  [3771] = {x=-41.457, y=32.468, z=44, rx=180, rz=-142.083, shoulder=lefty, elbow=epositive, wrist=wpositive, fatherId=fReference[0]}
  [3772] = {x=-40.218, y=31.503, z=44, rx=-180, rz=-142.07, shoulder=lefty, elbow=epositive, wrist=wpositive, fatherId=fReference[0]}
  [3773] = {x=-38.979, y=30.538, z=44, rx=-180, rz=-142.056, shoulder=lefty, elbow=epositive, wrist=wpositive, fatherId=fReference[0]}
  [3774] = {x=-37.74, y=29.572, z=44, rx=180, rz=-142.044, shoulder=lefty, elbow=epositive, wrist=wpositive, fatherId=fReference[0]}
  [3775] = {x=-36.502, y=28.606, z=44, rx=180, rz=-142.031, shoulder=lefty, elbow=epositive, wrist=wpositive, fatherId=fReference[0]}
  [3776] = {x=-35.263, y=27.639, z=44, rx=180, rz=-142.019, shoulder=lefty, elbow=epositive, wrist=wpositive, fatherId=fReference[0]}
  [3777] = {x=-34.025, y=26.672, z=44, rx=-180, rz=-142.007, shoulder=lefty, elbow=epositive, wrist=wpositive, fatherId=fReference[0]}
  [3778] = {x=-32.787, y=25.705, z=44, rx=-180, rz=-141.996, shoulder=lefty, elbow=epositive, wrist=wpositive, fatherId=fReference[0]}
  [3779] = {x=-31.549, y=24.738, z=44, rx=-180, rz=-141.985, shoulder=lefty, elbow=epositive, wrist=wpositive, fatherId=fReference[0]}
  [3780] = {x=-30.311, y=23.77, z=44, rx=180, rz=-141.975, shoulder=lefty, elbow=epositive, wrist=wpositive, fatherId=fReference[0]}
  [3781] = {x=-29.073, y=22.802, z=44, rx=-180, rz=-141.965, shoulder=lefty, elbow=epositive, wrist=wpositive, fatherId=fReference[0]}
  [3782] = {x=-27.835, y=21.834, z=44, rx=180, rz=-141.956, shoulder=lefty, elbow=epositive, wrist=wpositive, fatherId=fReference[0]}
  [3783] = {x=-26.597, y=20.865, z=44, rx=180, rz=-141.947, shoulder=lefty, elbow=epositive, wrist=wpositive, fatherId=fReference[0]}
  [3784] = {x=-25.36, y=19.896, z=44, rx=-180, rz=-141.938, shoulder=lefty, elbow=epositive, wrist=wpositive, fatherId=fReference[0]}
  [3785] = {x=-24.122, y=18.927, z=44, rx=-180, rz=-141.93, shoulder=lefty, elbow=epositive, wrist=wpositive, fatherId=fReference[0]}
  [3786] = {x=-22.885, y=17.958, z=44, rx=180, rz=-141.922, shoulder=lefty, elbow=epositive, wrist=wpositive, fatherId=fReference[0]}
  [3787] = {x=-21.647, y=16.988, z=44, rx=180, rz=-141.915, shoulder=lefty, elbow=epositive, wrist=wpositive, fatherId=fReference[0]}
  [3788] = {x=-20.41, y=16.019, z=44, rx=-180, rz=-141.908, shoulder=lefty, elbow=epositive, wrist=wpositive, fatherId=fReference[0]}
  [3789] = {x=-19.172, y=15.049, z=44, rx=-180, rz=-141.901, shoulder=lefty, elbow=epositive, wrist=wpositive, fatherId=fReference[0]}
  [3790] = {x=-17.935, y=14.079, z=44, rx=-180, rz=-141.895, shoulder=lefty, elbow=epositive, wrist=wpositive, fatherId=fReference[0]}
  [3791] = {x=-16.698, y=13.109, z=44, rx=180, rz=-141.889, shoulder=lefty, elbow=epositive, wrist=wpositive, fatherId=fReference[0]}
  [3792] = {x=-15.461, y=12.138, z=44, rx=-180, rz=-141.884, shoulder=lefty, elbow=epositive, wrist=wpositive, fatherId=fReference[0]}
  [3793] = {x=-14.224, y=11.168, z=44, rx=-180, rz=-141.879, shoulder=lefty, elbow=epositive, wrist=wpositive, fatherId=fReference[0]}
  [3794] = {x=-12.987, y=10.197, z=44, rx=-180, rz=-141.875, shoulder=lefty, elbow=epositive, wrist=wpositive, fatherId=fReference[0]}
  [3795] = {x=-11.75, y=9.226, z=44, rx=-180, rz=-141.871, shoulder=lefty, elbow=epositive, wrist=wpositive, fatherId=fReference[0]}
  [3796] = {x=-10.513, y=8.255, z=44, rx=180, rz=-141.867, shoulder=lefty, elbow=epositive, wrist=wpositive, fatherId=fReference[0]}
  [3797] = {x=-9.276, y=7.284, z=44, rx=-180, rz=-141.864, shoulder=lefty, elbow=epositive, wrist=wpositive, fatherId=fReference[0]}
  [3798] = {x=-8.039, y=6.313, z=44, rx=-180, rz=-141.862, shoulder=lefty, elbow=epositive, wrist=wpositive, fatherId=fReference[0]}
  [3799] = {x=-6.802, y=5.342, z=44, rx=-180, rz=-141.859, shoulder=lefty, elbow=epositive, wrist=wpositive, fatherId=fReference[0]}
  [3800] = {x=-5.565, y=4.37, z=44, rx=180, rz=-141.857, shoulder=lefty, elbow=epositive, wrist=wpositive, fatherId=fReference[0]}
  [3801] = {x=-4.328, y=3.399, z=44, rx=180, rz=-141.856, shoulder=lefty, elbow=epositive, wrist=wpositive, fatherId=fReference[0]}
  [3802] = {x=-3.091, y=2.427, z=44, rx=-180, rz=-141.855, shoulder=lefty, elbow=epositive, wrist=wpositive, fatherId=fReference[0]}
  [3803] = {x=-1.854, y=1.456, z=44, rx=180, rz=-141.854, shoulder=lefty, elbow=epositive, wrist=wpositive, fatherId=fReference[0]}
  [3804] = {x=-0.617, y=0.484, z=44, rx=180, rz=-141.854, shoulder=lefty, elbow=epositive, wrist=wpositive, fatherId=fReference[0]}
  [3805] = {x=0.62, y=-0.487, z=44, rx=-180, rz=-141.854, shoulder=lefty, elbow=epositive, wrist=wpositive, fatherId=fReference[0]}
  [3806] = {x=1.857, y=-1.459, z=44, rx=180, rz=-141.855, shoulder=lefty, elbow=epositive, wrist=wpositive, fatherId=fReference[0]}
  [3807] = {x=3.094, y=-2.43, z=44, rx=-180, rz=-141.856, shoulder=lefty, elbow=epositive, wrist=wpositive, fatherId=fReference[0]}
  [3808] = {x=4.331, y=-3.402, z=44, rx=180, rz=-141.857, shoulder=lefty, elbow=epositive, wrist=wpositive, fatherId=fReference[0]}
  [3809] = {x=5.568, y=-4.373, z=44, rx=-180, rz=-141.859, shoulder=lefty, elbow=epositive, wrist=wpositive, fatherId=fReference[0]}
  [3810] = {x=6.805, y=-5.345, z=44, rx=-180, rz=-141.862, shoulder=lefty, elbow=epositive, wrist=wpositive, fatherId=fReference[0]}
  [3811] = {x=8.043, y=-6.316, z=44, rx=-180, rz=-141.864, shoulder=lefty, elbow=epositive, wrist=wpositive, fatherId=fReference[0]}
  [3812] = {x=9.28, y=-7.287, z=44, rx=-180, rz=-141.867, shoulder=lefty, elbow=epositive, wrist=wpositive, fatherId=fReference[0]}
  [3813] = {x=10.517, y=-8.259, z=44, rx=180, rz=-141.871, shoulder=lefty, elbow=epositive, wrist=wpositive, fatherId=fReference[0]}
  [3814] = {x=11.754, y=-9.23, z=44, rx=180, rz=-141.875, shoulder=lefty, elbow=epositive, wrist=wpositive, fatherId=fReference[0]}
  [3815] = {x=12.992, y=-10.201, z=44, rx=-180, rz=-141.879, shoulder=lefty, elbow=epositive, wrist=wpositive, fatherId=fReference[0]}
  [3816] = {x=14.229, y=-11.172, z=44, rx=-180, rz=-141.884, shoulder=lefty, elbow=epositive, wrist=wpositive, fatherId=fReference[0]}
  [3817] = {x=15.467, y=-12.143, z=44, rx=-180, rz=-141.89, shoulder=lefty, elbow=epositive, wrist=wpositive, fatherId=fReference[0]}
  [3818] = {x=16.704, y=-13.113, z=44, rx=180, rz=-141.895, shoulder=lefty, elbow=epositive, wrist=wpositive, fatherId=fReference[0]}
  [3819] = {x=17.942, y=-14.084, z=44, rx=180, rz=-141.901, shoulder=lefty, elbow=epositive, wrist=wpositive, fatherId=fReference[0]}
  [3820] = {x=19.179, y=-15.054, z=44, rx=-180, rz=-141.908, shoulder=lefty, elbow=epositive, wrist=wpositive, fatherId=fReference[0]}
  [3821] = {x=20.417, y=-16.025, z=44, rx=180, rz=-141.915, shoulder=lefty, elbow=epositive, wrist=wpositive, fatherId=fReference[0]}
  [3822] = {x=21.655, y=-16.995, z=44, rx=-180, rz=-141.922, shoulder=lefty, elbow=epositive, wrist=wpositive, fatherId=fReference[0]}
  [3823] = {x=22.893, y=-17.965, z=44, rx=-180, rz=-141.93, shoulder=lefty, elbow=epositive, wrist=wpositive, fatherId=fReference[0]}
  [3824] = {x=24.131, y=-18.934, z=44, rx=-180, rz=-141.938, shoulder=lefty, elbow=epositive, wrist=wpositive, fatherId=fReference[0]}
  [3825] = {x=25.369, y=-19.904, z=44, rx=-180, rz=-141.947, shoulder=lefty, elbow=epositive, wrist=wpositive, fatherId=fReference[0]}
  [3826] = {x=26.607, y=-20.873, z=44, rx=180, rz=-141.956, shoulder=lefty, elbow=epositive, wrist=wpositive, fatherId=fReference[0]}
  [3827] = {x=27.846, y=-21.842, z=44, rx=-180, rz=-141.965, shoulder=lefty, elbow=epositive, wrist=wpositive, fatherId=fReference[0]}
  [3828] = {x=29.084, y=-22.811, z=44, rx=-180, rz=-141.975, shoulder=lefty, elbow=epositive, wrist=wpositive, fatherId=fReference[0]}
  [3829] = {x=30.323, y=-23.779, z=44, rx=180, rz=-141.986, shoulder=lefty, elbow=epositive, wrist=wpositive, fatherId=fReference[0]}
  [3830] = {x=31.561, y=-24.748, z=44, rx=-180, rz=-141.996, shoulder=lefty, elbow=epositive, wrist=wpositive, fatherId=fReference[0]}
  [3831] = {x=32.8, y=-25.716, z=44, rx=180, rz=-142.008, shoulder=lefty, elbow=epositive, wrist=wpositive, fatherId=fReference[0]}
  [3832] = {x=34.039, y=-26.683, z=44, rx=-180, rz=-142.019, shoulder=lefty, elbow=epositive, wrist=wpositive, fatherId=fReference[0]}
  [3833] = {x=35.278, y=-27.651, z=44, rx=-180, rz=-142.031, shoulder=lefty, elbow=epositive, wrist=wpositive, fatherId=fReference[0]}
  [3834] = {x=36.517, y=-28.618, z=44, rx=180, rz=-142.044, shoulder=lefty, elbow=epositive, wrist=wpositive, fatherId=fReference[0]}
  [3835] = {x=37.757, y=-29.585, z=44, rx=-180, rz=-142.057, shoulder=lefty, elbow=epositive, wrist=wpositive, fatherId=fReference[0]}
  [3836] = {x=38.996, y=-30.551, z=44, rx=-180, rz=-142.07, shoulder=lefty, elbow=epositive, wrist=wpositive, fatherId=fReference[0]}
  [3837] = {x=40.236, y=-31.517, z=44, rx=180, rz=-142.084, shoulder=lefty, elbow=epositive, wrist=wpositive, fatherId=fReference[0]}
  [3838] = {x=41.476, y=-32.483, z=44, rx=-180, rz=-142.098, shoulder=lefty, elbow=epositive, wrist=wpositive, fatherId=fReference[0]}
  [3839] = {x=42.715, y=-33.448, z=44, rx=-180, rz=-142.113, shoulder=lefty, elbow=epositive, wrist=wpositive, fatherId=fReference[0]}
  [3840] = {x=43.956, y=-34.413, z=44, rx=-180, rz=-142.128, shoulder=lefty, elbow=epositive, wrist=wpositive, fatherId=fReference[0]}
  [3841] = {x=45.196, y=-35.377, z=44, rx=180, rz=-142.143, shoulder=lefty, elbow=epositive, wrist=wpositive, fatherId=fReference[0]}
  [3842] = {x=46.436, y=-36.342, z=44, rx=-180, rz=-142.159, shoulder=lefty, elbow=epositive, wrist=wpositive, fatherId=fReference[0]}
  [3843] = {x=47.677, y=-37.305, z=44, rx=-180, rz=-142.175, shoulder=lefty, elbow=epositive, wrist=wpositive, fatherId=fReference[0]}
  [3844] = {x=48.917, y=-38.269, z=44, rx=180, rz=-142.192, shoulder=lefty, elbow=epositive, wrist=wpositive, fatherId=fReference[0]}
  [3845] = {x=50.158, y=-39.231, z=44, rx=-180, rz=-142.209, shoulder=lefty, elbow=epositive, wrist=wpositive, fatherId=fReference[0]}
  [3846] = {x=51.399, y=-40.194, z=44, rx=-180, rz=-142.227, shoulder=lefty, elbow=epositive, wrist=wpositive, fatherId=fReference[0]}
  [3847] = {x=52.641, y=-41.156, z=44, rx=-180, rz=-142.245, shoulder=lefty, elbow=epositive, wrist=wpositive, fatherId=fReference[0]}
  [3848] = {x=53.882, y=-42.117, z=44, rx=-180, rz=-142.263, shoulder=lefty, elbow=epositive, wrist=wpositive, fatherId=fReference[0]}
  [3849] = {x=55.124, y=-43.078, z=44, rx=180, rz=-142.282, shoulder=lefty, elbow=epositive, wrist=wpositive, fatherId=fReference[0]}
  [3850] = {x=56.366, y=-44.038, z=44, rx=-180, rz=-142.302, shoulder=lefty, elbow=epositive, wrist=wpositive, fatherId=fReference[0]}
  [3851] = {x=57.608, y=-44.998, z=44, rx=-180, rz=-142.321, shoulder=lefty, elbow=epositive, wrist=wpositive, fatherId=fReference[0]}
  [3852] = {x=58.85, y=-45.958, z=44, rx=-180, rz=-142.342, shoulder=lefty, elbow=epositive, wrist=wpositive, fatherId=fReference[0]}
  [3853] = {x=60.092, y=-46.916, z=44, rx=-180, rz=-142.362, shoulder=lefty, elbow=epositive, wrist=wpositive, fatherId=fReference[0]}
  [3854] = {x=61.335, y=-47.875, z=44, rx=-180, rz=-142.383, shoulder=lefty, elbow=epositive, wrist=wpositive, fatherId=fReference[0]}
  [3855] = {x=62.578, y=-48.832, z=44, rx=180, rz=-142.405, shoulder=lefty, elbow=epositive, wrist=wpositive, fatherId=fReference[0]}
  [3856] = {x=63.821, y=-49.79, z=44, rx=-180, rz=-142.427, shoulder=lefty, elbow=epositive, wrist=wpositive, fatherId=fReference[0]}
  [3857] = {x=65.064, y=-50.746, z=44, rx=-180, rz=-142.449, shoulder=lefty, elbow=epositive, wrist=wpositive, fatherId=fReference[0]}
  [3858] = {x=66.308, y=-51.702, z=44, rx=-180, rz=-142.472, shoulder=lefty, elbow=epositive, wrist=wpositive, fatherId=fReference[0]}
  [3859] = {x=67.551, y=-52.657, z=44, rx=-180, rz=-142.496, shoulder=lefty, elbow=epositive, wrist=wpositive, fatherId=fReference[0]}
  [3860] = {x=68.795, y=-53.612, z=44, rx=-180, rz=-142.519, shoulder=lefty, elbow=epositive, wrist=wpositive, fatherId=fReference[0]}
  [3861] = {x=70.04, y=-54.566, z=44, rx=-180, rz=-142.543, shoulder=lefty, elbow=epositive, wrist=wpositive, fatherId=fReference[0]}
  [3862] = {x=71.284, y=-55.519, z=44, rx=180, rz=-142.568, shoulder=lefty, elbow=epositive, wrist=wpositive, fatherId=fReference[0]}
  [3863] = {x=72.529, y=-56.472, z=44, rx=-180, rz=-142.593, shoulder=lefty, elbow=epositive, wrist=wpositive, fatherId=fReference[0]}
  [3864] = {x=73.774, y=-57.424, z=44, rx=180, rz=-142.619, shoulder=lefty, elbow=epositive, wrist=wpositive, fatherId=fReference[0]}
  [3865] = {x=75.019, y=-58.376, z=44, rx=-180, rz=-142.645, shoulder=lefty, elbow=epositive, wrist=wpositive, fatherId=fReference[0]}
  [3866] = {x=76.264, y=-59.326, z=44, rx=-180, rz=-142.671, shoulder=lefty, elbow=epositive, wrist=wpositive, fatherId=fReference[0]}
  [3867] = {x=77.51, y=-60.276, z=44, rx=-180, rz=-142.698, shoulder=lefty, elbow=epositive, wrist=wpositive, fatherId=fReference[0]}
  [3868] = {x=78.756, y=-61.226, z=44, rx=-180, rz=-142.725, shoulder=lefty, elbow=epositive, wrist=wpositive, fatherId=fReference[0]}
  [3869] = {x=80.002, y=-62.174, z=44, rx=180, rz=-142.753, shoulder=lefty, elbow=epositive, wrist=wpositive, fatherId=fReference[0]}
  [3870] = {x=81.249, y=-63.122, z=44, rx=180, rz=-142.781, shoulder=lefty, elbow=epositive, wrist=wpositive, fatherId=fReference[0]}
  [3871] = {x=82.496, y=-64.069, z=44, rx=180, rz=-142.81, shoulder=lefty, elbow=epositive, wrist=wpositive, fatherId=fReference[0]}
  [3872] = {x=83.743, y=-65.015, z=44, rx=-180, rz=-142.839, shoulder=lefty, elbow=epositive, wrist=wpositive, fatherId=fReference[0]}
  [3873] = {x=84.99, y=-65.961, z=44, rx=-180, rz=-142.868, shoulder=lefty, elbow=epositive, wrist=wpositive, fatherId=fReference[0]}
  [3874] = {x=86.238, y=-66.905, z=44, rx=180, rz=-142.898, shoulder=lefty, elbow=epositive, wrist=wpositive, fatherId=fReference[0]}
  [3875] = {x=87.486, y=-67.849, z=44, rx=-180, rz=-142.929, shoulder=lefty, elbow=epositive, wrist=wpositive, fatherId=fReference[0]}
  [3876] = {x=88.734, y=-68.792, z=44, rx=-180, rz=-142.96, shoulder=lefty, elbow=epositive, wrist=wpositive, fatherId=fReference[0]}
  [3877] = {x=89.982, y=-69.734, z=44, rx=-180, rz=-142.991, shoulder=lefty, elbow=epositive, wrist=wpositive, fatherId=fReference[0]}
  [3878] = {x=91.231, y=-70.676, z=44, rx=-180, rz=-143.023, shoulder=lefty, elbow=epositive, wrist=wpositive, fatherId=fReference[0]}
  [3879] = {x=92.48, y=-71.616, z=44, rx=180, rz=-143.055, shoulder=lefty, elbow=epositive, wrist=wpositive, fatherId=fReference[0]}
  [3880] = {x=93.73, y=-72.556, z=44, rx=-180, rz=-143.088, shoulder=lefty, elbow=epositive, wrist=wpositive, fatherId=fReference[0]}
  [3881] = {x=94.979, y=-73.495, z=44, rx=-180, rz=-143.121, shoulder=lefty, elbow=epositive, wrist=wpositive, fatherId=fReference[0]}
  [3882] = {x=96.23, y=-74.432, z=44, rx=-180, rz=-143.155, shoulder=lefty, elbow=epositive, wrist=wpositive, fatherId=fReference[0]}
  [3883] = {x=97.48, y=-75.369, z=44, rx=-180, rz=-143.189, shoulder=lefty, elbow=epositive, wrist=wpositive, fatherId=fReference[0]}
  [3884] = {x=98.731, y=-76.305, z=44, rx=-180, rz=-143.224, shoulder=lefty, elbow=epositive, wrist=wpositive, fatherId=fReference[0]}
  [3885] = {x=99.982, y=-77.24, z=44, rx=-180, rz=-143.259, shoulder=lefty, elbow=epositive, wrist=wpositive, fatherId=fReference[0]}
  [3886] = {x=101.233, y=-78.175, z=44, rx=-180, rz=-143.294, shoulder=lefty, elbow=epositive, wrist=wpositive, fatherId=fReference[0]}
  [3887] = {x=102.485, y=-79.108, z=44, rx=180, rz=-143.33, shoulder=lefty, elbow=epositive, wrist=wpositive, fatherId=fReference[0]}
  [3888] = {x=103.737, y=-80.04, z=44, rx=180, rz=-143.367, shoulder=lefty, elbow=epositive, wrist=wpositive, fatherId=fReference[0]}
  [3889] = {x=104.989, y=-80.971, z=44, rx=-180, rz=-143.404, shoulder=lefty, elbow=epositive, wrist=wpositive, fatherId=fReference[0]}
  [3890] = {x=106.242, y=-81.901, z=44, rx=180, rz=-143.441, shoulder=lefty, elbow=epositive, wrist=wpositive, fatherId=fReference[0]}
  [3891] = {x=107.495, y=-82.831, z=44, rx=-180, rz=-143.479, shoulder=lefty, elbow=epositive, wrist=wpositive, fatherId=fReference[0]}
  [3892] = {x=108.748, y=-83.759, z=44, rx=-180, rz=-143.517, shoulder=lefty, elbow=epositive, wrist=wpositive, fatherId=fReference[0]}
  [3893] = {x=110.002, y=-84.686, z=44, rx=-180, rz=-143.556, shoulder=lefty, elbow=epositive, wrist=wpositive, fatherId=fReference[0]}
  [3894] = {x=111.256, y=-85.612, z=44, rx=-180, rz=-143.596, shoulder=lefty, elbow=epositive, wrist=wpositive, fatherId=fReference[0]}
  [3895] = {x=112.511, y=-86.537, z=44, rx=-180, rz=-143.635, shoulder=lefty, elbow=epositive, wrist=wpositive, fatherId=fReference[0]}
  [3896] = {x=113.766, y=-87.461, z=44, rx=-180, rz=-143.676, shoulder=lefty, elbow=epositive, wrist=wpositive, fatherId=fReference[0]}
  [3897] = {x=115.021, y=-88.384, z=44, rx=180, rz=-143.716, shoulder=lefty, elbow=epositive, wrist=wpositive, fatherId=fReference[0]}
  [3898] = {x=116.277, y=-89.306, z=44, rx=-180, rz=-143.758, shoulder=lefty, elbow=epositive, wrist=wpositive, fatherId=fReference[0]}
  [3899] = {x=117.533, y=-90.227, z=44, rx=-180, rz=-143.799, shoulder=lefty, elbow=epositive, wrist=wpositive, fatherId=fReference[0]}
  [3900] = {x=118.789, y=-91.146, z=44, rx=180, rz=-143.842, shoulder=lefty, elbow=epositive, wrist=wpositive, fatherId=fReference[0]}
  [3901] = {x=120.046, y=-92.065, z=44, rx=-180, rz=-143.884, shoulder=lefty, elbow=epositive, wrist=wpositive, fatherId=fReference[0]}
  [3902] = {x=121.304, y=-92.982, z=44, rx=-180, rz=-143.927, shoulder=lefty, elbow=epositive, wrist=wpositive, fatherId=fReference[0]}
  [3903] = {x=122.561, y=-93.898, z=44, rx=-180, rz=-143.971, shoulder=lefty, elbow=epositive, wrist=wpositive, fatherId=fReference[0]}
  [3904] = {x=123.819, y=-94.813, z=44, rx=-180, rz=-144.015, shoulder=lefty, elbow=epositive, wrist=wpositive, fatherId=fReference[0]}
  [3905] = {x=125.078, y=-95.727, z=44, rx=180, rz=-144.06, shoulder=lefty, elbow=epositive, wrist=wpositive, fatherId=fReference[0]}
  [3906] = {x=126.337, y=-96.64, z=44, rx=180, rz=-144.105, shoulder=lefty, elbow=epositive, wrist=wpositive, fatherId=fReference[0]}
  [3907] = {x=127.596, y=-97.551, z=44, rx=-180, rz=-144.151, shoulder=lefty, elbow=epositive, wrist=wpositive, fatherId=fReference[0]}
  [3908] = {x=128.856, y=-98.461, z=44, rx=180, rz=-144.197, shoulder=lefty, elbow=epositive, wrist=wpositive, fatherId=fReference[0]}
  [3909] = {x=130.116, y=-99.37, z=44, rx=-180, rz=-144.243, shoulder=lefty, elbow=epositive, wrist=wpositive, fatherId=fReference[0]}
  [3910] = {x=131.376, y=-100.278, z=44, rx=-180, rz=-144.291, shoulder=lefty, elbow=epositive, wrist=wpositive, fatherId=fReference[0]}
  [3911] = {x=132.637, y=-101.185, z=44, rx=-180, rz=-144.338, shoulder=lefty, elbow=epositive, wrist=wpositive, fatherId=fReference[0]}
  [3912] = {x=133.899, y=-102.09, z=44, rx=180, rz=-144.386, shoulder=lefty, elbow=epositive, wrist=wpositive, fatherId=fReference[0]}
  [3913] = {x=135.161, y=-102.994, z=44, rx=-180, rz=-144.435, shoulder=lefty, elbow=epositive, wrist=wpositive, fatherId=fReference[0]}
  [3914] = {x=136.423, y=-103.896, z=44, rx=-180, rz=-144.484, shoulder=lefty, elbow=epositive, wrist=wpositive, fatherId=fReference[0]}
  [3915] = {x=137.686, y=-104.798, z=44, rx=-180, rz=-144.534, shoulder=lefty, elbow=epositive, wrist=wpositive, fatherId=fReference[0]}
  [3916] = {x=138.949, y=-105.698, z=44, rx=-180, rz=-144.584, shoulder=lefty, elbow=epositive, wrist=wpositive, fatherId=fReference[0]}
  [3917] = {x=140.213, y=-106.596, z=44, rx=-180, rz=-144.634, shoulder=lefty, elbow=epositive, wrist=wpositive, fatherId=fReference[0]}
  [3918] = {x=141.477, y=-107.494, z=44, rx=180, rz=-144.686, shoulder=lefty, elbow=epositive, wrist=wpositive, fatherId=fReference[0]}
  [3919] = {x=142.742, y=-108.389, z=44, rx=-180, rz=-144.737, shoulder=lefty, elbow=epositive, wrist=wpositive, fatherId=fReference[0]}
  [3920] = {x=144.007, y=-109.284, z=44, rx=-180, rz=-144.789, shoulder=lefty, elbow=epositive, wrist=wpositive, fatherId=fReference[0]}
  [3921] = {x=145.273, y=-110.177, z=44, rx=180, rz=-144.842, shoulder=lefty, elbow=epositive, wrist=wpositive, fatherId=fReference[0]}
  [3922] = {x=146.539, y=-111.069, z=44, rx=-180, rz=-144.895, shoulder=lefty, elbow=epositive, wrist=wpositive, fatherId=fReference[0]}
  [3923] = {x=147.806, y=-111.959, z=44, rx=180, rz=-144.949, shoulder=lefty, elbow=epositive, wrist=wpositive, fatherId=fReference[0]}
  [3924] = {x=149.073, y=-112.848, z=44, rx=-180, rz=-145.003, shoulder=lefty, elbow=epositive, wrist=wpositive, fatherId=fReference[0]}
  [3925] = {x=150.34, y=-113.736, z=44, rx=-180, rz=-145.058, shoulder=lefty, elbow=epositive, wrist=wpositive, fatherId=fReference[0]}
  [3926] = {x=151.608, y=-114.622, z=44, rx=-180, rz=-145.113, shoulder=lefty, elbow=epositive, wrist=wpositive, fatherId=fReference[0]}
  [3927] = {x=152.877, y=-115.506, z=44, rx=-180, rz=-145.169, shoulder=lefty, elbow=epositive, wrist=wpositive, fatherId=fReference[0]}
  [3928] = {x=154.146, y=-116.389, z=44, rx=180, rz=-145.225, shoulder=lefty, elbow=epositive, wrist=wpositive, fatherId=fReference[0]}
  [3929] = {x=155.416, y=-117.271, z=44, rx=180, rz=-145.282, shoulder=lefty, elbow=epositive, wrist=wpositive, fatherId=fReference[0]}
  [3930] = {x=156.686, y=-118.151, z=44, rx=-180, rz=-145.34, shoulder=lefty, elbow=epositive, wrist=wpositive, fatherId=fReference[0]}
  [3931] = {x=157.957, y=-119.03, z=44, rx=-180, rz=-145.398, shoulder=lefty, elbow=epositive, wrist=wpositive, fatherId=fReference[0]}
  [3932] = {x=159.228, y=-119.907, z=44, rx=180, rz=-145.456, shoulder=lefty, elbow=epositive, wrist=wpositive, fatherId=fReference[0]}
  [3933] = {x=160.5, y=-120.782, z=44, rx=-180, rz=-145.515, shoulder=lefty, elbow=epositive, wrist=wpositive, fatherId=fReference[0]}
  [3934] = {x=161.772, y=-121.656, z=44, rx=180, rz=-145.575, shoulder=lefty, elbow=epositive, wrist=wpositive, fatherId=fReference[0]}
  [3935] = {x=163.045, y=-122.529, z=44, rx=180, rz=-145.635, shoulder=lefty, elbow=epositive, wrist=wpositive, fatherId=fReference[0]}
  [3936] = {x=164.319, y=-123.4, z=44, rx=180, rz=-145.695, shoulder=lefty, elbow=epositive, wrist=wpositive, fatherId=fReference[0]}
  [3937] = {x=165.593, y=-124.269, z=44, rx=-180, rz=-145.756, shoulder=lefty, elbow=epositive, wrist=wpositive, fatherId=fReference[0]}
  [3938] = {x=166.867, y=-125.136, z=44, rx=-180, rz=-145.818, shoulder=lefty, elbow=epositive, wrist=wpositive, fatherId=fReference[0]}
  [3939] = {x=168.142, y=-126.002, z=44, rx=-180, rz=-145.88, shoulder=lefty, elbow=epositive, wrist=wpositive, fatherId=fReference[0]}
  [3940] = {x=169.418, y=-126.867, z=44, rx=180, rz=-145.943, shoulder=lefty, elbow=epositive, wrist=wpositive, fatherId=fReference[0]}
  [3941] = {x=170.695, y=-127.73, z=44, rx=-180, rz=-146.006, shoulder=lefty, elbow=epositive, wrist=wpositive, fatherId=fReference[0]}
  [3942] = {x=171.971, y=-128.591, z=44, rx=-180, rz=-146.07, shoulder=lefty, elbow=epositive, wrist=wpositive, fatherId=fReference[0]}
  [3943] = {x=173.249, y=-129.45, z=44, rx=180, rz=-146.135, shoulder=lefty, elbow=epositive, wrist=wpositive, fatherId=fReference[0]}
  [3944] = {x=174.527, y=-130.308, z=44, rx=180, rz=-146.2, shoulder=lefty, elbow=epositive, wrist=wpositive, fatherId=fReference[0]}
  [3945] = {x=175.806, y=-131.164, z=44, rx=-180, rz=-146.265, shoulder=lefty, elbow=epositive, wrist=wpositive, fatherId=fReference[0]}
  [3946] = {x=177.085, y=-132.018, z=44, rx=-180, rz=-146.331, shoulder=lefty, elbow=epositive, wrist=wpositive, fatherId=fReference[0]}
  [3947] = {x=178.365, y=-132.871, z=44, rx=180, rz=-146.398, shoulder=lefty, elbow=epositive, wrist=wpositive, fatherId=fReference[0]}
  [3948] = {x=179.645, y=-133.721, z=44, rx=-180, rz=-146.465, shoulder=lefty, elbow=epositive, wrist=wpositive, fatherId=fReference[0]}
  [3949] = {x=180.927, y=-134.571, z=44, rx=-180, rz=-146.533, shoulder=lefty, elbow=epositive, wrist=wpositive, fatherId=fReference[0]}
  [3950] = {x=182.208, y=-135.418, z=44, rx=-180, rz=-146.601, shoulder=lefty, elbow=epositive, wrist=wpositive, fatherId=fReference[0]}
  [3951] = {x=183.491, y=-136.263, z=44, rx=180, rz=-146.67, shoulder=lefty, elbow=epositive, wrist=wpositive, fatherId=fReference[0]}
  [3952] = {x=184.774, y=-137.107, z=44, rx=-180, rz=-146.74, shoulder=lefty, elbow=epositive, wrist=wpositive, fatherId=fReference[0]}
  [3953] = {x=186.057, y=-137.949, z=44, rx=-180, rz=-146.81, shoulder=lefty, elbow=epositive, wrist=wpositive, fatherId=fReference[0]}
  [3954] = {x=187.341, y=-138.789, z=44, rx=180, rz=-146.881, shoulder=lefty, elbow=epositive, wrist=wpositive, fatherId=fReference[0]}
  [3955] = {x=188.626, y=-139.627, z=44, rx=-180, rz=-146.952, shoulder=lefty, elbow=epositive, wrist=wpositive, fatherId=fReference[0]}
  [3956] = {x=189.912, y=-140.464, z=44, rx=-180, rz=-147.024, shoulder=lefty, elbow=epositive, wrist=wpositive, fatherId=fReference[0]}
  [3957] = {x=191.198, y=-141.298, z=44, rx=-180, rz=-147.096, shoulder=lefty, elbow=epositive, wrist=wpositive, fatherId=fReference[0]}
  [3958] = {x=192.485, y=-142.131, z=44, rx=-180, rz=-147.169, shoulder=lefty, elbow=epositive, wrist=wpositive, fatherId=fReference[0]}
  [3959] = {x=193.772, y=-142.961, z=44, rx=-180, rz=-147.243, shoulder=lefty, elbow=epositive, wrist=wpositive, fatherId=fReference[0]}
  [3960] = {x=195.06, y=-143.79, z=44, rx=-180, rz=-147.317, shoulder=lefty, elbow=epositive, wrist=wpositive, fatherId=fReference[0]}
  [3961] = {x=196.349, y=-144.617, z=44, rx=-180, rz=-147.392, shoulder=lefty, elbow=epositive, wrist=wpositive, fatherId=fReference[0]}
  [3962] = {x=197.639, y=-145.442, z=44, rx=-180, rz=-147.467, shoulder=lefty, elbow=epositive, wrist=wpositive, fatherId=fReference[0]}
  [3963] = {x=198.929, y=-146.265, z=44, rx=-180, rz=-147.543, shoulder=lefty, elbow=epositive, wrist=wpositive, fatherId=fReference[0]}
  [3964] = {x=200.219, y=-147.086, z=44, rx=-180, rz=-147.619, shoulder=lefty, elbow=epositive, wrist=wpositive, fatherId=fReference[0]}
  [3965] = {x=201.511, y=-147.905, z=44, rx=-180, rz=-147.697, shoulder=lefty, elbow=epositive, wrist=wpositive, fatherId=fReference[0]}
  [3966] = {x=202.803, y=-148.722, z=44, rx=-180, rz=-147.774, shoulder=lefty, elbow=epositive, wrist=wpositive, fatherId=fReference[0]}
  [3967] = {x=204.096, y=-149.536, z=44, rx=-180, rz=-147.853, shoulder=lefty, elbow=epositive, wrist=wpositive, fatherId=fReference[0]}
  [3968] = {x=205.389, y=-150.349, z=44, rx=-180, rz=-147.931, shoulder=lefty, elbow=epositive, wrist=wpositive, fatherId=fReference[0]}
  [3969] = {x=206.683, y=-151.16, z=44, rx=180, rz=-148.011, shoulder=lefty, elbow=epositive, wrist=wpositive, fatherId=fReference[0]}
  [3970] = {x=207.978, y=-151.969, z=44, rx=180, rz=-148.091, shoulder=lefty, elbow=epositive, wrist=wpositive, fatherId=fReference[0]}
  [3971] = {x=209.273, y=-152.775, z=44, rx=180, rz=-148.172, shoulder=lefty, elbow=epositive, wrist=wpositive, fatherId=fReference[0]}
  [3972] = {x=210.569, y=-153.58, z=44, rx=180, rz=-148.253, shoulder=lefty, elbow=epositive, wrist=wpositive, fatherId=fReference[0]}
  [3973] = {x=211.866, y=-154.382, z=44, rx=180, rz=-148.335, shoulder=lefty, elbow=epositive, wrist=wpositive, fatherId=fReference[0]}
  [3974] = {x=213.164, y=-155.183, z=44, rx=-180, rz=-148.418, shoulder=lefty, elbow=epositive, wrist=wpositive, fatherId=fReference[0]}
  [3975] = {x=214.462, y=-155.981, z=44, rx=-180, rz=-148.501, shoulder=lefty, elbow=epositive, wrist=wpositive, fatherId=fReference[0]}
  [3976] = {x=215.761, y=-156.777, z=44, rx=180, rz=-148.585, shoulder=lefty, elbow=epositive, wrist=wpositive, fatherId=fReference[0]}
  [3977] = {x=217.06, y=-157.57, z=44, rx=-180, rz=-148.669, shoulder=lefty, elbow=epositive, wrist=wpositive, fatherId=fReference[0]}
  [3978] = {x=218.361, y=-158.362, z=44, rx=-180, rz=-148.754, shoulder=lefty, elbow=epositive, wrist=wpositive, fatherId=fReference[0]}
  [3979] = {x=219.662, y=-159.151, z=44, rx=180, rz=-148.84, shoulder=lefty, elbow=epositive, wrist=wpositive, fatherId=fReference[0]}
  [3980] = {x=220.963, y=-159.938, z=44, rx=-180, rz=-148.926, shoulder=lefty, elbow=epositive, wrist=wpositive, fatherId=fReference[0]}
  [3981] = {x=222.266, y=-160.723, z=44, rx=-180, rz=-149.013, shoulder=lefty, elbow=epositive, wrist=wpositive, fatherId=fReference[0]}
  [3982] = {x=223.569, y=-161.506, z=44, rx=180, rz=-149.101, shoulder=lefty, elbow=epositive, wrist=wpositive, fatherId=fReference[0]}
  [3983] = {x=224.872, y=-162.286, z=44, rx=180, rz=-149.189, shoulder=lefty, elbow=epositive, wrist=wpositive, fatherId=fReference[0]}
  [3984] = {x=226.177, y=-163.064, z=44, rx=-180, rz=-149.278, shoulder=lefty, elbow=epositive, wrist=wpositive, fatherId=fReference[0]}
  [3985] = {x=227.482, y=-163.84, z=44, rx=-180, rz=-149.367, shoulder=lefty, elbow=epositive, wrist=wpositive, fatherId=fReference[0]}
  [3986] = {x=228.788, y=-164.613, z=44, rx=-180, rz=-149.458, shoulder=lefty, elbow=epositive, wrist=wpositive, fatherId=fReference[0]}
  [3987] = {x=230.095, y=-165.384, z=44, rx=-180, rz=-149.548, shoulder=lefty, elbow=epositive, wrist=wpositive, fatherId=fReference[0]}
  [3988] = {x=231.402, y=-166.152, z=44, rx=-180, rz=-149.64, shoulder=lefty, elbow=epositive, wrist=wpositive, fatherId=fReference[0]}
  [3989] = {x=232.71, y=-166.919, z=44, rx=-180, rz=-149.732, shoulder=lefty, elbow=epositive, wrist=wpositive, fatherId=fReference[0]}
  [3990] = {x=234.019, y=-167.682, z=44, rx=-180, rz=-149.824, shoulder=lefty, elbow=epositive, wrist=wpositive, fatherId=fReference[0]}
  [3991] = {x=235.328, y=-168.444, z=44, rx=-180, rz=-149.918, shoulder=lefty, elbow=epositive, wrist=wpositive, fatherId=fReference[0]}
  [3992] = {x=236.638, y=-169.203, z=44, rx=-180, rz=-150.012, shoulder=lefty, elbow=epositive, wrist=wpositive, fatherId=fReference[0]}
  [3993] = {x=237.949, y=-169.959, z=44, rx=-180, rz=-150.106, shoulder=lefty, elbow=epositive, wrist=wpositive, fatherId=fReference[0]}
  [3994] = {x=239.261, y=-170.713, z=44, rx=-180, rz=-150.202, shoulder=lefty, elbow=epositive, wrist=wpositive, fatherId=fReference[0]}
  [3995] = {x=240.573, y=-171.465, z=44, rx=-180, rz=-150.298, shoulder=lefty, elbow=epositive, wrist=wpositive, fatherId=fReference[0]}
  [3996] = {x=241.886, y=-172.214, z=44, rx=-180, rz=-150.394, shoulder=lefty, elbow=epositive, wrist=wpositive, fatherId=fReference[0]}
  [3997] = {x=243.2, y=-172.96, z=44, rx=-180, rz=-150.491, shoulder=lefty, elbow=epositive, wrist=wpositive, fatherId=fReference[0]}
  [3998] = {x=244.514, y=-173.704, z=44, rx=-180, rz=-150.589, shoulder=lefty, elbow=epositive, wrist=wpositive, fatherId=fReference[0]}
  [3999] = {x=245.83, y=-174.446, z=44, rx=-180, rz=-150.688, shoulder=lefty, elbow=epositive, wrist=wpositive, fatherId=fReference[0]}
  [4000] = {x=247.146, y=-175.184, z=44, rx=-180, rz=-150.787, shoulder=lefty, elbow=epositive, wrist=wpositive, fatherId=fReference[0]}
  [4001] = {x=248.462, y=-175.921, z=44, rx=180, rz=-150.887, shoulder=lefty, elbow=epositive, wrist=wpositive, fatherId=fReference[0]}
  [4002] = {x=249.78, y=-176.654, z=44, rx=-180, rz=-150.988, shoulder=lefty, elbow=epositive, wrist=wpositive, fatherId=fReference[0]}
  [4003] = {x=251.098, y=-177.385, z=44, rx=180, rz=-151.089, shoulder=lefty, elbow=epositive, wrist=wpositive, fatherId=fReference[0]}
  [4004] = {x=252.417, y=-178.114, z=44, rx=-180, rz=-151.191, shoulder=lefty, elbow=epositive, wrist=wpositive, fatherId=fReference[0]}
  [4005] = {x=253.736, y=-178.839, z=44, rx=-180, rz=-151.293, shoulder=lefty, elbow=epositive, wrist=wpositive, fatherId=fReference[0]}
  [4006] = {x=255.056, y=-179.562, z=44, rx=180, rz=-151.397, shoulder=lefty, elbow=epositive, wrist=wpositive, fatherId=fReference[0]}
  [4007] = {x=256.378, y=-180.283, z=44, rx=180, rz=-151.501, shoulder=lefty, elbow=epositive, wrist=wpositive, fatherId=fReference[0]}
  [4008] = {x=257.699, y=-181, z=44, rx=-180, rz=-151.605, shoulder=lefty, elbow=epositive, wrist=wpositive, fatherId=fReference[0]}
  [4009] = {x=259.022, y=-181.715, z=44, rx=180, rz=-151.711, shoulder=lefty, elbow=epositive, wrist=wpositive, fatherId=fReference[0]}
  [4010] = {x=260.345, y=-182.427, z=44, rx=-180, rz=-151.817, shoulder=lefty, elbow=epositive, wrist=wpositive, fatherId=fReference[0]}
  [4011] = {x=261.669, y=-183.137, z=44, rx=-180, rz=-151.923, shoulder=lefty, elbow=epositive, wrist=wpositive, fatherId=fReference[0]}
  [4012] = {x=262.994, y=-183.843, z=44, rx=180, rz=-152.031, shoulder=lefty, elbow=epositive, wrist=wpositive, fatherId=fReference[0]}
  [4013] = {x=264.319, y=-184.547, z=44, rx=-180, rz=-152.139, shoulder=lefty, elbow=epositive, wrist=wpositive, fatherId=fReference[0]}
  [4014] = {x=265.645, y=-185.248, z=44, rx=-180, rz=-152.247, shoulder=lefty, elbow=epositive, wrist=wpositive, fatherId=fReference[0]}
  [4015] = {x=266.972, y=-185.946, z=44, rx=180, rz=-152.357, shoulder=lefty, elbow=epositive, wrist=wpositive, fatherId=fReference[0]}
  [4016] = {x=268.3, y=-186.642, z=44, rx=180, rz=-152.467, shoulder=lefty, elbow=epositive, wrist=wpositive, fatherId=fReference[0]}
  [4017] = {x=269.628, y=-187.334, z=44, rx=180, rz=-152.578, shoulder=lefty, elbow=epositive, wrist=wpositive, fatherId=fReference[0]}
  [4018] = {x=270.957, y=-188.024, z=44, rx=-180, rz=-152.689, shoulder=lefty, elbow=epositive, wrist=wpositive, fatherId=fReference[0]}
  [4019] = {x=272.287, y=-188.711, z=44, rx=-180, rz=-152.801, shoulder=lefty, elbow=epositive, wrist=wpositive, fatherId=fReference[0]}
  [4020] = {x=273.617, y=-189.394, z=44, rx=180, rz=-152.914, shoulder=lefty, elbow=epositive, wrist=wpositive, fatherId=fReference[0]}
  [4021] = {x=274.948, y=-190.075, z=44, rx=-180, rz=-153.028, shoulder=lefty, elbow=epositive, wrist=wpositive, fatherId=fReference[0]}
  [4022] = {x=276.28, y=-190.753, z=44, rx=-180, rz=-153.142, shoulder=lefty, elbow=epositive, wrist=wpositive, fatherId=fReference[0]}
  [4023] = {x=277.613, y=-191.428, z=44, rx=-180, rz=-153.257, shoulder=lefty, elbow=epositive, wrist=wpositive, fatherId=fReference[0]}
  [4024] = {x=278.947, y=-192.1, z=44, rx=-180, rz=-153.372, shoulder=lefty, elbow=epositive, wrist=wpositive, fatherId=fReference[0]}
  [4025] = {x=280.281, y=-192.769, z=44, rx=-180, rz=-153.489, shoulder=lefty, elbow=epositive, wrist=wpositive, fatherId=fReference[0]}
  [4026] = {x=281.616, y=-193.435, z=44, rx=-180, rz=-153.606, shoulder=lefty, elbow=epositive, wrist=wpositive, fatherId=fReference[0]}
  [4027] = {x=282.951, y=-194.097, z=44, rx=-180, rz=-153.724, shoulder=lefty, elbow=epositive, wrist=wpositive, fatherId=fReference[0]}
  [4028] = {x=284.288, y=-194.757, z=44, rx=180, rz=-153.842, shoulder=lefty, elbow=epositive, wrist=wpositive, fatherId=fReference[0]}
  [4029] = {x=285.625, y=-195.414, z=44, rx=-180, rz=-153.961, shoulder=lefty, elbow=epositive, wrist=wpositive, fatherId=fReference[0]}
  [4030] = {x=286.963, y=-196.068, z=44, rx=180, rz=-154.081, shoulder=lefty, elbow=epositive, wrist=wpositive, fatherId=fReference[0]}
  [4031] = {x=288.301, y=-196.718, z=44, rx=-180, rz=-154.202, shoulder=lefty, elbow=epositive, wrist=wpositive, fatherId=fReference[0]}
  [4032] = {x=289.64, y=-197.365, z=44, rx=-180, rz=-154.323, shoulder=lefty, elbow=epositive, wrist=wpositive, fatherId=fReference[0]}
  [4033] = {x=290.98, y=-198.01, z=44, rx=180, rz=-154.445, shoulder=lefty, elbow=epositive, wrist=wpositive, fatherId=fReference[0]}
  [4034] = {x=292.321, y=-198.651, z=44, rx=-180, rz=-154.568, shoulder=lefty, elbow=epositive, wrist=wpositive, fatherId=fReference[0]}
  [4035] = {x=293.663, y=-199.289, z=44, rx=-180, rz=-154.691, shoulder=lefty, elbow=epositive, wrist=wpositive, fatherId=fReference[0]}
  [4036] = {x=295.005, y=-199.923, z=44, rx=-180, rz=-154.815, shoulder=lefty, elbow=epositive, wrist=wpositive, fatherId=fReference[0]}
  [4037] = {x=296.348, y=-200.555, z=44, rx=-180, rz=-154.94, shoulder=lefty, elbow=epositive, wrist=wpositive, fatherId=fReference[0]}
  [4038] = {x=297.691, y=-201.183, z=44, rx=-180, rz=-155.066, shoulder=lefty, elbow=epositive, wrist=wpositive, fatherId=fReference[0]}
  [4039] = {x=299.036, y=-201.808, z=44, rx=180, rz=-155.192, shoulder=lefty, elbow=epositive, wrist=wpositive, fatherId=fReference[0]}
  [4040] = {x=300.381, y=-202.43, z=44, rx=-180, rz=-155.319, shoulder=lefty, elbow=epositive, wrist=wpositive, fatherId=fReference[0]}
  [4041] = {x=301.727, y=-203.048, z=44, rx=-180, rz=-155.447, shoulder=lefty, elbow=epositive, wrist=wpositive, fatherId=fReference[0]}
  [4042] = {x=303.073, y=-203.663, z=44, rx=-180, rz=-155.575, shoulder=lefty, elbow=epositive, wrist=wpositive, fatherId=fReference[0]}
  [4043] = {x=304.421, y=-204.275, z=44, rx=-180, rz=-155.705, shoulder=lefty, elbow=epositive, wrist=wpositive, fatherId=fReference[0]}
  [4044] = {x=305.769, y=-204.884, z=44, rx=180, rz=-155.835, shoulder=lefty, elbow=epositive, wrist=wpositive, fatherId=fReference[0]}
  [4045] = {x=307.117, y=-205.489, z=44, rx=-180, rz=-155.965, shoulder=lefty, elbow=epositive, wrist=wpositive, fatherId=fReference[0]}
  [4046] = {x=308.467, y=-206.091, z=44, rx=-180, rz=-156.097, shoulder=lefty, elbow=epositive, wrist=wpositive, fatherId=fReference[0]}
  [4047] = {x=309.817, y=-206.689, z=44, rx=180, rz=-156.229, shoulder=lefty, elbow=epositive, wrist=wpositive, fatherId=fReference[0]}
  [4048] = {x=311.168, y=-207.284, z=44, rx=-180, rz=-156.361, shoulder=lefty, elbow=epositive, wrist=wpositive, fatherId=fReference[0]}
  [4049] = {x=312.519, y=-207.876, z=44, rx=180, rz=-156.495, shoulder=lefty, elbow=epositive, wrist=wpositive, fatherId=fReference[0]}
  [4050] = {x=313.872, y=-208.464, z=44, rx=180, rz=-156.629, shoulder=lefty, elbow=epositive, wrist=wpositive, fatherId=fReference[0]}
  [4051] = {x=315.225, y=-209.049, z=44, rx=-180, rz=-156.764, shoulder=lefty, elbow=epositive, wrist=wpositive, fatherId=fReference[0]}
  [4052] = {x=316.579, y=-209.63, z=44, rx=-180, rz=-156.9, shoulder=lefty, elbow=epositive, wrist=wpositive, fatherId=fReference[0]}
  [4053] = {x=317.933, y=-210.208, z=44, rx=-180, rz=-157.036, shoulder=lefty, elbow=epositive, wrist=wpositive, fatherId=fReference[0]}
  [4054] = {x=319.288, y=-210.782, z=44, rx=180, rz=-157.173, shoulder=lefty, elbow=epositive, wrist=wpositive, fatherId=fReference[0]}
  [4055] = {x=320.644, y=-211.353, z=44, rx=180, rz=-157.311, shoulder=lefty, elbow=epositive, wrist=wpositive, fatherId=fReference[0]}
  [4056] = {x=322.001, y=-211.92, z=44, rx=-180, rz=-157.45, shoulder=lefty, elbow=epositive, wrist=wpositive, fatherId=fReference[0]}
  [4057] = {x=323.358, y=-212.483, z=44, rx=-180, rz=-157.589, shoulder=lefty, elbow=epositive, wrist=wpositive, fatherId=fReference[0]}
  [4058] = {x=324.716, y=-213.044, z=44, rx=180, rz=-157.729, shoulder=lefty, elbow=epositive, wrist=wpositive, fatherId=fReference[0]}
  [4059] = {x=326.075, y=-213.6, z=44, rx=180, rz=-157.87, shoulder=lefty, elbow=epositive, wrist=wpositive, fatherId=fReference[0]}
  [4060] = {x=327.435, y=-214.153, z=44, rx=-180, rz=-158.011, shoulder=lefty, elbow=epositive, wrist=wpositive, fatherId=fReference[0]}
  [4061] = {x=328.795, y=-214.702, z=44, rx=180, rz=-158.153, shoulder=lefty, elbow=epositive, wrist=wpositive, fatherId=fReference[0]}
  [4062] = {x=330.156, y=-215.248, z=44, rx=180, rz=-158.296, shoulder=lefty, elbow=epositive, wrist=wpositive, fatherId=fReference[0]}
  [4063] = {x=331.517, y=-215.79, z=44, rx=-180, rz=-158.44, shoulder=lefty, elbow=epositive, wrist=wpositive, fatherId=fReference[0]}
  [4064] = {x=332.88, y=-216.328, z=44, rx=-180, rz=-158.584, shoulder=lefty, elbow=epositive, wrist=wpositive, fatherId=fReference[0]}
  [4065] = {x=334.243, y=-216.863, z=44, rx=-180, rz=-158.729, shoulder=lefty, elbow=epositive, wrist=wpositive, fatherId=fReference[0]}
  [4066] = {x=335.607, y=-217.394, z=44, rx=180, rz=-158.875, shoulder=lefty, elbow=epositive, wrist=wpositive, fatherId=fReference[0]}
  [4067] = {x=336.971, y=-217.921, z=44, rx=-180, rz=-159.022, shoulder=lefty, elbow=epositive, wrist=wpositive, fatherId=fReference[0]}
  [4068] = {x=338.336, y=-218.444, z=44, rx=180, rz=-159.169, shoulder=lefty, elbow=epositive, wrist=wpositive, fatherId=fReference[0]}
  [4069] = {x=339.702, y=-218.964, z=44, rx=-180, rz=-159.317, shoulder=lefty, elbow=epositive, wrist=wpositive, fatherId=fReference[0]}
  [4070] = {x=341.069, y=-219.48, z=44, rx=-180, rz=-159.465, shoulder=lefty, elbow=epositive, wrist=wpositive, fatherId=fReference[0]}
  [4071] = {x=342.436, y=-219.992, z=44, rx=-180, rz=-159.615, shoulder=lefty, elbow=epositive, wrist=wpositive, fatherId=fReference[0]}
  [4072] = {x=343.804, y=-220.5, z=44, rx=-180, rz=-159.765, shoulder=lefty, elbow=epositive, wrist=wpositive, fatherId=fReference[0]}
  [4073] = {x=345.173, y=-221.005, z=44, rx=-180, rz=-159.916, shoulder=lefty, elbow=epositive, wrist=wpositive, fatherId=fReference[0]}
  [4074] = {x=346.542, y=-221.506, z=44, rx=-180, rz=-160.067, shoulder=lefty, elbow=epositive, wrist=wpositive, fatherId=fReference[0]}
  [4075] = {x=347.912, y=-222.002, z=44, rx=-180, rz=-160.219, shoulder=lefty, elbow=epositive, wrist=wpositive, fatherId=fReference[0]}
  [4076] = {x=349.283, y=-222.495, z=44, rx=-180, rz=-160.372, shoulder=lefty, elbow=epositive, wrist=wpositive, fatherId=fReference[0]}
  [4077] = {x=350.655, y=-222.985, z=44, rx=-180, rz=-160.526, shoulder=lefty, elbow=epositive, wrist=wpositive, fatherId=fReference[0]}
  [4078] = {x=352.027, y=-223.47, z=44, rx=-180, rz=-160.68, shoulder=lefty, elbow=epositive, wrist=wpositive, fatherId=fReference[0]}
  [4079] = {x=353.4, y=-223.951, z=44, rx=180, rz=-160.835, shoulder=lefty, elbow=epositive, wrist=wpositive, fatherId=fReference[0]}
  [4080] = {x=354.773, y=-224.429, z=44, rx=-180, rz=-160.991, shoulder=lefty, elbow=epositive, wrist=wpositive, fatherId=fReference[0]}
  [4081] = {x=356.148, y=-224.902, z=44, rx=-180, rz=-161.147, shoulder=lefty, elbow=epositive, wrist=wpositive, fatherId=fReference[0]}
  [4082] = {x=357.523, y=-225.371, z=44, rx=-180, rz=-161.304, shoulder=lefty, elbow=epositive, wrist=wpositive, fatherId=fReference[0]}
  [4083] = {x=358.898, y=-225.837, z=44, rx=180, rz=-161.462, shoulder=lefty, elbow=epositive, wrist=wpositive, fatherId=fReference[0]}
  [4084] = {x=360.275, y=-226.298, z=44, rx=-180, rz=-161.621, shoulder=lefty, elbow=epositive, wrist=wpositive, fatherId=fReference[0]}
  [4085] = {x=361.652, y=-226.756, z=44, rx=180, rz=-161.78, shoulder=lefty, elbow=epositive, wrist=wpositive, fatherId=fReference[0]}
  [4086] = {x=363.029, y=-227.209, z=44, rx=-180, rz=-161.94, shoulder=lefty, elbow=epositive, wrist=wpositive, fatherId=fReference[0]}
  [4087] = {x=364.407, y=-227.659, z=44, rx=180, rz=-162.1, shoulder=lefty, elbow=epositive, wrist=wpositive, fatherId=fReference[0]}
  [4088] = {x=365.786, y=-228.104, z=44, rx=-180, rz=-162.262, shoulder=lefty, elbow=epositive, wrist=wpositive, fatherId=fReference[0]}
  [4089] = {x=367.166, y=-228.546, z=44, rx=-180, rz=-162.424, shoulder=lefty, elbow=epositive, wrist=wpositive, fatherId=fReference[0]}
  [4090] = {x=368.546, y=-228.983, z=44, rx=-180, rz=-162.586, shoulder=lefty, elbow=epositive, wrist=wpositive, fatherId=fReference[0]}
  [4091] = {x=369.927, y=-229.416, z=44, rx=180, rz=-162.75, shoulder=lefty, elbow=epositive, wrist=wpositive, fatherId=fReference[0]}
  [4092] = {x=371.309, y=-229.845, z=44, rx=180, rz=-162.913, shoulder=lefty, elbow=epositive, wrist=wpositive, fatherId=fReference[0]}
  [4093] = {x=372.691, y=-230.27, z=44, rx=-180, rz=-163.078, shoulder=lefty, elbow=epositive, wrist=wpositive, fatherId=fReference[0]}
  [4094] = {x=374.074, y=-230.69, z=44, rx=-180, rz=-163.243, shoulder=lefty, elbow=epositive, wrist=wpositive, fatherId=fReference[0]}
  [4095] = {x=375.457, y=-231.107, z=44, rx=-180, rz=-163.409, shoulder=lefty, elbow=epositive, wrist=wpositive, fatherId=fReference[0]}
  [4096] = {x=376.841, y=-231.519, z=44, rx=-180, rz=-163.576, shoulder=lefty, elbow=epositive, wrist=wpositive, fatherId=fReference[0]}
  [4097] = {x=378.226, y=-231.928, z=44, rx=-180, rz=-163.743, shoulder=lefty, elbow=epositive, wrist=wpositive, fatherId=fReference[0]}
  [4098] = {x=379.611, y=-232.331, z=44, rx=-180, rz=-163.911, shoulder=lefty, elbow=epositive, wrist=wpositive, fatherId=fReference[0]}
  [4099] = {x=380.997, y=-232.731, z=44, rx=-180, rz=-164.08, shoulder=lefty, elbow=epositive, wrist=wpositive, fatherId=fReference[0]}
  [4100] = {x=382.384, y=-233.127, z=44, rx=-180, rz=-164.249, shoulder=lefty, elbow=epositive, wrist=wpositive, fatherId=fReference[0]}
  [4101] = {x=383.771, y=-233.518, z=44, rx=180, rz=-164.419, shoulder=lefty, elbow=epositive, wrist=wpositive, fatherId=fReference[0]}
  [4102] = {x=385.159, y=-233.905, z=44, rx=-180, rz=-164.589, shoulder=lefty, elbow=epositive, wrist=wpositive, fatherId=fReference[0]}
  [4103] = {x=386.547, y=-234.288, z=44, rx=180, rz=-164.76, shoulder=lefty, elbow=epositive, wrist=wpositive, fatherId=fReference[0]}
  [4104] = {x=387.936, y=-234.666, z=44, rx=-180, rz=-164.932, shoulder=lefty, elbow=epositive, wrist=wpositive, fatherId=fReference[0]}
  [4105] = {x=389.325, y=-235.04, z=44, rx=-180, rz=-165.105, shoulder=lefty, elbow=epositive, wrist=wpositive, fatherId=fReference[0]}
  [4106] = {x=390.715, y=-235.41, z=44, rx=180, rz=-165.277, shoulder=lefty, elbow=epositive, wrist=wpositive, fatherId=fReference[0]}
  [4107] = {x=392.106, y=-235.775, z=44, rx=180, rz=-165.451, shoulder=lefty, elbow=epositive, wrist=wpositive, fatherId=fReference[0]}
  [4108] = {x=393.497, y=-236.136, z=44, rx=-180, rz=-165.625, shoulder=lefty, elbow=epositive, wrist=wpositive, fatherId=fReference[0]}
  [4109] = {x=394.889, y=-236.493, z=44, rx=180, rz=-165.8, shoulder=lefty, elbow=epositive, wrist=wpositive, fatherId=fReference[0]}
  [4110] = {x=396.281, y=-236.845, z=44, rx=-180, rz=-165.976, shoulder=lefty, elbow=epositive, wrist=wpositive, fatherId=fReference[0]}
  [4111] = {x=397.674, y=-237.193, z=44, rx=180, rz=-166.152, shoulder=lefty, elbow=epositive, wrist=wpositive, fatherId=fReference[0]}
  [4112] = {x=399.068, y=-237.537, z=44, rx=180, rz=-166.328, shoulder=lefty, elbow=epositive, wrist=wpositive, fatherId=fReference[0]}
  [4113] = {x=400.462, y=-237.876, z=44, rx=180, rz=-166.505, shoulder=lefty, elbow=epositive, wrist=wpositive, fatherId=fReference[0]}
  [4114] = {x=401.856, y=-238.21, z=44, rx=-180, rz=-166.683, shoulder=lefty, elbow=epositive, wrist=wpositive, fatherId=fReference[0]}
  [4115] = {x=403.251, y=-238.541, z=44, rx=-180, rz=-166.861, shoulder=lefty, elbow=epositive, wrist=wpositive, fatherId=fReference[0]}
  [4116] = {x=404.647, y=-238.866, z=44, rx=-180, rz=-167.04, shoulder=lefty, elbow=epositive, wrist=wpositive, fatherId=fReference[0]}
  [4117] = {x=406.043, y=-239.188, z=44, rx=-180, rz=-167.22, shoulder=lefty, elbow=epositive, wrist=wpositive, fatherId=fReference[0]}
  [4118] = {x=407.439, y=-239.505, z=44, rx=180, rz=-167.4, shoulder=lefty, elbow=epositive, wrist=wpositive, fatherId=fReference[0]}
  [4119] = {x=408.836, y=-239.817, z=44, rx=180, rz=-167.581, shoulder=lefty, elbow=epositive, wrist=wpositive, fatherId=fReference[0]}
  [4120] = {x=410.234, y=-240.125, z=44, rx=180, rz=-167.762, shoulder=lefty, elbow=epositive, wrist=wpositive, fatherId=fReference[0]}
  [4121] = {x=411.632, y=-240.428, z=44, rx=180, rz=-167.943, shoulder=lefty, elbow=epositive, wrist=wpositive, fatherId=fReference[0]}
  [4122] = {x=413.031, y=-240.727, z=44, rx=180, rz=-168.126, shoulder=lefty, elbow=epositive, wrist=wpositive, fatherId=fReference[0]}
  [4123] = {x=414.43, y=-241.021, z=44, rx=-180, rz=-168.308, shoulder=lefty, elbow=epositive, wrist=wpositive, fatherId=fReference[0]}
  [4124] = {x=415.829, y=-241.31, z=44, rx=180, rz=-168.492, shoulder=lefty, elbow=epositive, wrist=wpositive, fatherId=fReference[0]}
  [4125] = {x=417.229, y=-241.595, z=44, rx=-180, rz=-168.675, shoulder=lefty, elbow=epositive, wrist=wpositive, fatherId=fReference[0]}
  [4126] = {x=418.63, y=-241.876, z=44, rx=-180, rz=-168.86, shoulder=lefty, elbow=epositive, wrist=wpositive, fatherId=fReference[0]}
  [4127] = {x=420.031, y=-242.152, z=44, rx=180, rz=-169.045, shoulder=lefty, elbow=epositive, wrist=wpositive, fatherId=fReference[0]}
  [4128] = {x=421.432, y=-242.423, z=44, rx=-180, rz=-169.23, shoulder=lefty, elbow=epositive, wrist=wpositive, fatherId=fReference[0]}
  [4129] = {x=422.834, y=-242.69, z=44, rx=180, rz=-169.416, shoulder=lefty, elbow=epositive, wrist=wpositive, fatherId=fReference[0]}
  [4130] = {x=424.236, y=-242.952, z=44, rx=180, rz=-169.602, shoulder=lefty, elbow=epositive, wrist=wpositive, fatherId=fReference[0]}
  [4131] = {x=425.639, y=-243.209, z=44, rx=180, rz=-169.789, shoulder=lefty, elbow=epositive, wrist=wpositive, fatherId=fReference[0]}
  [4132] = {x=427.042, y=-243.462, z=44, rx=180, rz=-169.976, shoulder=lefty, elbow=epositive, wrist=wpositive, fatherId=fReference[0]}
  [4133] = {x=428.445, y=-243.71, z=44, rx=-180, rz=-170.164, shoulder=lefty, elbow=epositive, wrist=wpositive, fatherId=fReference[0]}
  [4134] = {x=429.849, y=-243.953, z=44, rx=-180, rz=-170.352, shoulder=lefty, elbow=epositive, wrist=wpositive, fatherId=fReference[0]}
  [4135] = {x=431.254, y=-244.192, z=44, rx=-180, rz=-170.54, shoulder=lefty, elbow=epositive, wrist=wpositive, fatherId=fReference[0]}
  [4136] = {x=432.658, y=-244.426, z=44, rx=180, rz=-170.729, shoulder=lefty, elbow=epositive, wrist=wpositive, fatherId=fReference[0]}
  [4137] = {x=434.064, y=-244.655, z=44, rx=180, rz=-170.919, shoulder=lefty, elbow=epositive, wrist=wpositive, fatherId=fReference[0]}
  [4138] = {x=435.469, y=-244.88, z=44, rx=180, rz=-171.109, shoulder=lefty, elbow=epositive, wrist=wpositive, fatherId=fReference[0]}
  [4139] = {x=436.875, y=-245.1, z=44, rx=-180, rz=-171.299, shoulder=lefty, elbow=epositive, wrist=wpositive, fatherId=fReference[0]}
  [4140] = {x=438.281, y=-245.315, z=44, rx=-180, rz=-171.49, shoulder=lefty, elbow=epositive, wrist=wpositive, fatherId=fReference[0]}
  [4141] = {x=439.688, y=-245.526, z=44, rx=180, rz=-171.681, shoulder=lefty, elbow=epositive, wrist=wpositive, fatherId=fReference[0]}
  [4142] = {x=441.095, y=-245.731, z=44, rx=180, rz=-171.873, shoulder=lefty, elbow=epositive, wrist=wpositive, fatherId=fReference[0]}
  [4143] = {x=442.502, y=-245.932, z=44, rx=180, rz=-172.065, shoulder=lefty, elbow=epositive, wrist=wpositive, fatherId=fReference[0]}
  [4144] = {x=443.91, y=-246.129, z=44, rx=-180, rz=-172.257, shoulder=lefty, elbow=epositive, wrist=wpositive, fatherId=fReference[0]}
  [4145] = {x=445.318, y=-246.32, z=44, rx=-180, rz=-172.449, shoulder=lefty, elbow=epositive, wrist=wpositive, fatherId=fReference[0]}
  [4146] = {x=446.726, y=-246.507, z=44, rx=180, rz=-172.643, shoulder=lefty, elbow=epositive, wrist=wpositive, fatherId=fReference[0]}
  [4147] = {x=448.134, y=-246.689, z=44, rx=-180, rz=-172.836, shoulder=lefty, elbow=epositive, wrist=wpositive, fatherId=fReference[0]}
  [4148] = {x=449.543, y=-246.866, z=44, rx=180, rz=-173.03, shoulder=lefty, elbow=epositive, wrist=wpositive, fatherId=fReference[0]}
  [4149] = {x=450.953, y=-247.038, z=44, rx=-180, rz=-173.224, shoulder=lefty, elbow=epositive, wrist=wpositive, fatherId=fReference[0]}
  [4150] = {x=452.362, y=-247.205, z=44, rx=-180, rz=-173.418, shoulder=lefty, elbow=epositive, wrist=wpositive, fatherId=fReference[0]}
  [4151] = {x=453.772, y=-247.368, z=44, rx=-180, rz=-173.613, shoulder=lefty, elbow=epositive, wrist=wpositive, fatherId=fReference[0]}
  [4152] = {x=455.182, y=-247.526, z=44, rx=-180, rz=-173.808, shoulder=lefty, elbow=epositive, wrist=wpositive, fatherId=fReference[0]}
  [4153] = {x=456.592, y=-247.679, z=44, rx=180, rz=-174.003, shoulder=lefty, elbow=epositive, wrist=wpositive, fatherId=fReference[0]}
  [4154] = {x=458.003, y=-247.827, z=44, rx=-180, rz=-174.199, shoulder=lefty, elbow=epositive, wrist=wpositive, fatherId=fReference[0]}
  [4155] = {x=459.414, y=-247.971, z=44, rx=180, rz=-174.395, shoulder=lefty, elbow=epositive, wrist=wpositive, fatherId=fReference[0]}
  [4156] = {x=460.825, y=-248.109, z=44, rx=-180, rz=-174.591, shoulder=lefty, elbow=epositive, wrist=wpositive, fatherId=fReference[0]}
  [4157] = {x=462.236, y=-248.243, z=44, rx=180, rz=-174.787, shoulder=lefty, elbow=epositive, wrist=wpositive, fatherId=fReference[0]}
  [4158] = {x=463.647, y=-248.371, z=44, rx=180, rz=-174.984, shoulder=lefty, elbow=epositive, wrist=wpositive, fatherId=fReference[0]}
  [4159] = {x=465.059, y=-248.495, z=44, rx=-180, rz=-175.181, shoulder=lefty, elbow=epositive, wrist=wpositive, fatherId=fReference[0]}
  [4160] = {x=466.471, y=-248.614, z=44, rx=-180, rz=-175.378, shoulder=lefty, elbow=epositive, wrist=wpositive, fatherId=fReference[0]}
  [4161] = {x=467.883, y=-248.729, z=44, rx=-180, rz=-175.575, shoulder=lefty, elbow=epositive, wrist=wpositive, fatherId=fReference[0]}
  [4162] = {x=469.296, y=-248.838, z=44, rx=-180, rz=-175.773, shoulder=lefty, elbow=epositive, wrist=wpositive, fatherId=fReference[0]}
  [4163] = {x=470.708, y=-248.942, z=44, rx=180, rz=-175.971, shoulder=lefty, elbow=epositive, wrist=wpositive, fatherId=fReference[0]}
  [4164] = {x=472.121, y=-249.042, z=44, rx=180, rz=-176.169, shoulder=lefty, elbow=epositive, wrist=wpositive, fatherId=fReference[0]}
  [4165] = {x=473.534, y=-249.136, z=44, rx=-180, rz=-176.367, shoulder=lefty, elbow=epositive, wrist=wpositive, fatherId=fReference[0]}
  [4166] = {x=474.947, y=-249.226, z=44, rx=-180, rz=-176.566, shoulder=lefty, elbow=epositive, wrist=wpositive, fatherId=fReference[0]}
  [4167] = {x=476.36, y=-249.311, z=44, rx=180, rz=-176.764, shoulder=lefty, elbow=epositive, wrist=wpositive, fatherId=fReference[0]}
  [4168] = {x=477.773, y=-249.391, z=44, rx=180, rz=-176.963, shoulder=lefty, elbow=epositive, wrist=wpositive, fatherId=fReference[0]}
  [4169] = {x=479.187, y=-249.466, z=44, rx=-180, rz=-177.162, shoulder=lefty, elbow=epositive, wrist=wpositive, fatherId=fReference[0]}
  [4170] = {x=480.6, y=-249.536, z=44, rx=-180, rz=-177.361, shoulder=lefty, elbow=epositive, wrist=wpositive, fatherId=fReference[0]}
  [4171] = {x=482.014, y=-249.601, z=44, rx=-180, rz=-177.56, shoulder=lefty, elbow=epositive, wrist=wpositive, fatherId=fReference[0]}
  [4172] = {x=483.428, y=-249.661, z=44, rx=180, rz=-177.759, shoulder=lefty, elbow=epositive, wrist=wpositive, fatherId=fReference[0]}
  [4173] = {x=484.841, y=-249.717, z=44, rx=-180, rz=-177.959, shoulder=lefty, elbow=epositive, wrist=wpositive, fatherId=fReference[0]}
  [4174] = {x=486.255, y=-249.767, z=44, rx=180, rz=-178.158, shoulder=lefty, elbow=epositive, wrist=wpositive, fatherId=fReference[0]}
  [4175] = {x=487.669, y=-249.812, z=44, rx=-180, rz=-178.358, shoulder=lefty, elbow=epositive, wrist=wpositive, fatherId=fReference[0]}
  [4176] = {x=489.084, y=-249.853, z=44, rx=-180, rz=-178.557, shoulder=lefty, elbow=epositive, wrist=wpositive, fatherId=fReference[0]}
  [4177] = {x=490.498, y=-249.889, z=44, rx=180, rz=-178.757, shoulder=lefty, elbow=epositive, wrist=wpositive, fatherId=fReference[0]}
  [4178] = {x=491.912, y=-249.919, z=44, rx=-180, rz=-178.957, shoulder=lefty, elbow=epositive, wrist=wpositive, fatherId=fReference[0]}
  [4179] = {x=493.326, y=-249.945, z=44, rx=-180, rz=-179.157, shoulder=lefty, elbow=epositive, wrist=wpositive, fatherId=fReference[0]}
  [4180] = {x=494.741, y=-249.966, z=44, rx=-180, rz=-179.357, shoulder=lefty, elbow=epositive, wrist=wpositive, fatherId=fReference[0]}
  [4181] = {x=496.155, y=-249.982, z=44, rx=180, rz=-179.557, shoulder=lefty, elbow=epositive, wrist=wpositive, fatherId=fReference[0]}
  [4182] = {x=497.569, y=-249.993, z=44, rx=-180, rz=-179.756, shoulder=lefty, elbow=epositive, wrist=wpositive, fatherId=fReference[0]}
  [4183] = {x=498.984, y=-249.999, z=44, rx=-180, rz=-179.956, shoulder=lefty, elbow=epositive, wrist=wpositive, fatherId=fReference[0]}
  [4184] = {x=500.398, y=-250, z=44, rx=-180, rz=179.844, shoulder=lefty, elbow=epositive, wrist=wpositive, fatherId=fReference[0]}
  [4185] = {x=501.812, y=-249.996, z=44, rx=-180, rz=179.644, shoulder=lefty, elbow=epositive, wrist=wpositive, fatherId=fReference[0]}
  [4186] = {x=503.227, y=-249.987, z=44, rx=-180, rz=179.444, shoulder=lefty, elbow=epositive, wrist=wpositive, fatherId=fReference[0]}
  [4187] = {x=504.641, y=-249.973, z=44, rx=180, rz=179.244, shoulder=lefty, elbow=epositive, wrist=wpositive, fatherId=fReference[0]}
  [4188] = {x=506.055, y=-249.955, z=44, rx=-180, rz=179.044, shoulder=lefty, elbow=epositive, wrist=wpositive, fatherId=fReference[0]}
  [4189] = {x=507.47, y=-249.931, z=44, rx=-180, rz=178.844, shoulder=lefty, elbow=epositive, wrist=wpositive, fatherId=fReference[0]}
  [4190] = {x=508.884, y=-249.903, z=44, rx=180, rz=178.645, shoulder=lefty, elbow=epositive, wrist=wpositive, fatherId=fReference[0]}
  [4191] = {x=510.298, y=-249.869, z=44, rx=-180, rz=178.445, shoulder=lefty, elbow=epositive, wrist=wpositive, fatherId=fReference[0]}
  [4192] = {x=511.712, y=-249.831, z=44, rx=180, rz=178.245, shoulder=lefty, elbow=epositive, wrist=wpositive, fatherId=fReference[0]}
  [4193] = {x=513.126, y=-249.787, z=44, rx=-180, rz=178.046, shoulder=lefty, elbow=epositive, wrist=wpositive, fatherId=fReference[0]}
  [4194] = {x=514.54, y=-249.739, z=44, rx=180, rz=177.846, shoulder=lefty, elbow=epositive, wrist=wpositive, fatherId=fReference[0]}
  [4195] = {x=515.954, y=-249.686, z=44, rx=180, rz=177.647, shoulder=lefty, elbow=epositive, wrist=wpositive, fatherId=fReference[0]}
  [4196] = {x=517.368, y=-249.628, z=44, rx=-180, rz=177.448, shoulder=lefty, elbow=epositive, wrist=wpositive, fatherId=fReference[0]}
  [4197] = {x=518.782, y=-249.565, z=44, rx=180, rz=177.249, shoulder=lefty, elbow=epositive, wrist=wpositive, fatherId=fReference[0]}
  [4198] = {x=520.195, y=-249.497, z=44, rx=-180, rz=177.05, shoulder=lefty, elbow=epositive, wrist=wpositive, fatherId=fReference[0]}
  [4199] = {x=521.609, y=-249.424, z=44, rx=180, rz=176.851, shoulder=lefty, elbow=epositive, wrist=wpositive, fatherId=fReference[0]}
  [4200] = {x=523.022, y=-249.346, z=44, rx=180, rz=176.652, shoulder=lefty, elbow=epositive, wrist=wpositive, fatherId=fReference[0]}
  [4201] = {x=524.435, y=-249.264, z=44, rx=180, rz=176.454, shoulder=lefty, elbow=epositive, wrist=wpositive, fatherId=fReference[0]}
  [4202] = {x=525.848, y=-249.176, z=44, rx=-180, rz=176.256, shoulder=lefty, elbow=epositive, wrist=wpositive, fatherId=fReference[0]}
  [4203] = {x=527.261, y=-249.084, z=44, rx=180, rz=176.058, shoulder=lefty, elbow=epositive, wrist=wpositive, fatherId=fReference[0]}
  [4204] = {x=528.674, y=-248.986, z=44, rx=-180, rz=175.86, shoulder=lefty, elbow=epositive, wrist=wpositive, fatherId=fReference[0]}
  [4205] = {x=530.086, y=-248.884, z=44, rx=-180, rz=175.662, shoulder=lefty, elbow=epositive, wrist=wpositive, fatherId=fReference[0]}
  [4206] = {x=531.498, y=-248.777, z=44, rx=-180, rz=175.465, shoulder=lefty, elbow=epositive, wrist=wpositive, fatherId=fReference[0]}
  [4207] = {x=532.911, y=-248.665, z=44, rx=-180, rz=175.267, shoulder=lefty, elbow=epositive, wrist=wpositive, fatherId=fReference[0]}
  [4208] = {x=534.323, y=-248.548, z=44, rx=180, rz=175.07, shoulder=lefty, elbow=epositive, wrist=wpositive, fatherId=fReference[0]}
  [4209] = {x=535.734, y=-248.426, z=44, rx=-180, rz=174.874, shoulder=lefty, elbow=epositive, wrist=wpositive, fatherId=fReference[0]}
  [4210] = {x=537.146, y=-248.3, z=44, rx=-180, rz=174.677, shoulder=lefty, elbow=epositive, wrist=wpositive, fatherId=fReference[0]}
  [4211] = {x=538.557, y=-248.168, z=44, rx=-180, rz=174.481, shoulder=lefty, elbow=epositive, wrist=wpositive, fatherId=fReference[0]}
  [4212] = {x=539.968, y=-248.032, z=44, rx=-180, rz=174.285, shoulder=lefty, elbow=epositive, wrist=wpositive, fatherId=fReference[0]}
  [4213] = {x=541.379, y=-247.891, z=44, rx=-180, rz=174.089, shoulder=lefty, elbow=epositive, wrist=wpositive, fatherId=fReference[0]}
  [4214] = {x=542.79, y=-247.744, z=44, rx=180, rz=173.894, shoulder=lefty, elbow=epositive, wrist=wpositive, fatherId=fReference[0]}
  [4215] = {x=544.2, y=-247.594, z=44, rx=180, rz=173.698, shoulder=lefty, elbow=epositive, wrist=wpositive, fatherId=fReference[0]}
  [4216] = {x=545.61, y=-247.438, z=44, rx=180, rz=173.504, shoulder=lefty, elbow=epositive, wrist=wpositive, fatherId=fReference[0]}
  [4217] = {x=547.02, y=-247.277, z=44, rx=-180, rz=173.309, shoulder=lefty, elbow=epositive, wrist=wpositive, fatherId=fReference[0]}
  [4218] = {x=548.43, y=-247.112, z=44, rx=-180, rz=173.115, shoulder=lefty, elbow=epositive, wrist=wpositive, fatherId=fReference[0]}
  [4219] = {x=549.839, y=-246.942, z=44, rx=-180, rz=172.921, shoulder=lefty, elbow=epositive, wrist=wpositive, fatherId=fReference[0]}
  [4220] = {x=551.248, y=-246.767, z=44, rx=180, rz=172.727, shoulder=lefty, elbow=epositive, wrist=wpositive, fatherId=fReference[0]}
  [4221] = {x=552.657, y=-246.587, z=44, rx=180, rz=172.534, shoulder=lefty, elbow=epositive, wrist=wpositive, fatherId=fReference[0]}
  [4222] = {x=554.065, y=-246.402, z=44, rx=-180, rz=172.341, shoulder=lefty, elbow=epositive, wrist=wpositive, fatherId=fReference[0]}
  [4223] = {x=555.473, y=-246.213, z=44, rx=180, rz=172.149, shoulder=lefty, elbow=epositive, wrist=wpositive, fatherId=fReference[0]}
  [4224] = {x=556.881, y=-246.019, z=44, rx=180, rz=171.957, shoulder=lefty, elbow=epositive, wrist=wpositive, fatherId=fReference[0]}
  [4225] = {x=558.289, y=-245.82, z=44, rx=-180, rz=171.765, shoulder=lefty, elbow=epositive, wrist=wpositive, fatherId=fReference[0]}
  [4226] = {x=559.696, y=-245.616, z=44, rx=-180, rz=171.574, shoulder=lefty, elbow=epositive, wrist=wpositive, fatherId=fReference[0]}
  [4227] = {x=561.102, y=-245.408, z=44, rx=180, rz=171.383, shoulder=lefty, elbow=epositive, wrist=wpositive, fatherId=fReference[0]}
  [4228] = {x=562.509, y=-245.195, z=44, rx=-180, rz=171.192, shoulder=lefty, elbow=epositive, wrist=wpositive, fatherId=fReference[0]}
  [4229] = {x=563.915, y=-244.977, z=44, rx=180, rz=171.002, shoulder=lefty, elbow=epositive, wrist=wpositive, fatherId=fReference[0]}
  [4230] = {x=565.321, y=-244.755, z=44, rx=-180, rz=170.813, shoulder=lefty, elbow=epositive, wrist=wpositive, fatherId=fReference[0]}
  [4231] = {x=566.726, y=-244.527, z=44, rx=-180, rz=170.623, shoulder=lefty, elbow=epositive, wrist=wpositive, fatherId=fReference[0]}
  [4232] = {x=568.131, y=-244.295, z=44, rx=-180, rz=170.435, shoulder=lefty, elbow=epositive, wrist=wpositive, fatherId=fReference[0]}
  [4233] = {x=569.535, y=-244.059, z=44, rx=-180, rz=170.246, shoulder=lefty, elbow=epositive, wrist=wpositive, fatherId=fReference[0]}
  [4234] = {x=570.939, y=-243.817, z=44, rx=-180, rz=170.058, shoulder=lefty, elbow=epositive, wrist=wpositive, fatherId=fReference[0]}
  [4235] = {x=572.343, y=-243.571, z=44, rx=-180, rz=169.871, shoulder=lefty, elbow=epositive, wrist=wpositive, fatherId=fReference[0]}
  [4236] = {x=573.746, y=-243.32, z=44, rx=-180, rz=169.684, shoulder=lefty, elbow=epositive, wrist=wpositive, fatherId=fReference[0]}
  [4237] = {x=575.149, y=-243.065, z=44, rx=-180, rz=169.497, shoulder=lefty, elbow=epositive, wrist=wpositive, fatherId=fReference[0]}
  [4238] = {x=576.552, y=-242.805, z=44, rx=-180, rz=169.311, shoulder=lefty, elbow=epositive, wrist=wpositive, fatherId=fReference[0]}
  [4239] = {x=577.954, y=-242.54, z=44, rx=180, rz=169.126, shoulder=lefty, elbow=epositive, wrist=wpositive, fatherId=fReference[0]}
  [4240] = {x=579.355, y=-242.271, z=44, rx=180, rz=168.941, shoulder=lefty, elbow=epositive, wrist=wpositive, fatherId=fReference[0]}
  [4241] = {x=580.757, y=-241.997, z=44, rx=-180, rz=168.756, shoulder=lefty, elbow=epositive, wrist=wpositive, fatherId=fReference[0]}
  [4242] = {x=582.157, y=-241.719, z=44, rx=180, rz=168.572, shoulder=lefty, elbow=epositive, wrist=wpositive, fatherId=fReference[0]}
  [4243] = {x=583.557, y=-241.436, z=44, rx=180, rz=168.389, shoulder=lefty, elbow=epositive, wrist=wpositive, fatherId=fReference[0]}
  [4244] = {x=584.957, y=-241.148, z=44, rx=-180, rz=168.206, shoulder=lefty, elbow=epositive, wrist=wpositive, fatherId=fReference[0]}
  [4245] = {x=586.357, y=-240.856, z=44, rx=-180, rz=168.023, shoulder=lefty, elbow=epositive, wrist=wpositive, fatherId=fReference[0]}
  [4246] = {x=587.755, y=-240.559, z=44, rx=-180, rz=167.841, shoulder=lefty, elbow=epositive, wrist=wpositive, fatherId=fReference[0]}
  [4247] = {x=589.154, y=-240.258, z=44, rx=-180, rz=167.66, shoulder=lefty, elbow=epositive, wrist=wpositive, fatherId=fReference[0]}
  [4248] = {x=590.552, y=-239.952, z=44, rx=180, rz=167.479, shoulder=lefty, elbow=epositive, wrist=wpositive, fatherId=fReference[0]}
  [4249] = {x=591.949, y=-239.642, z=44, rx=-180, rz=167.299, shoulder=lefty, elbow=epositive, wrist=wpositive, fatherId=fReference[0]}
  [4250] = {x=593.346, y=-239.327, z=44, rx=180, rz=167.119, shoulder=lefty, elbow=epositive, wrist=wpositive, fatherId=fReference[0]}
  [4251] = {x=594.742, y=-239.008, z=44, rx=-180, rz=166.94, shoulder=lefty, elbow=epositive, wrist=wpositive, fatherId=fReference[0]}
  [4252] = {x=596.138, y=-238.684, z=44, rx=180, rz=166.761, shoulder=lefty, elbow=epositive, wrist=wpositive, fatherId=fReference[0]}
  [4253] = {x=597.533, y=-238.356, z=44, rx=180, rz=166.583, shoulder=lefty, elbow=epositive, wrist=wpositive, fatherId=fReference[0]}
  [4254] = {x=598.928, y=-238.023, z=44, rx=180, rz=166.405, shoulder=lefty, elbow=epositive, wrist=wpositive, fatherId=fReference[0]}
  [4255] = {x=600.322, y=-237.686, z=44, rx=180, rz=166.229, shoulder=lefty, elbow=epositive, wrist=wpositive, fatherId=fReference[0]}
  [4256] = {x=601.716, y=-237.344, z=44, rx=-180, rz=166.052, shoulder=lefty, elbow=epositive, wrist=wpositive, fatherId=fReference[0]}
  [4257] = {x=603.109, y=-236.998, z=44, rx=180, rz=165.877, shoulder=lefty, elbow=epositive, wrist=wpositive, fatherId=fReference[0]}
  [4258] = {x=604.502, y=-236.648, z=44, rx=-180, rz=165.702, shoulder=lefty, elbow=epositive, wrist=wpositive, fatherId=fReference[0]}
  [4259] = {x=605.894, y=-236.293, z=44, rx=180, rz=165.527, shoulder=lefty, elbow=epositive, wrist=wpositive, fatherId=fReference[0]}
  [4260] = {x=607.286, y=-235.934, z=44, rx=-180, rz=165.353, shoulder=lefty, elbow=epositive, wrist=wpositive, fatherId=fReference[0]}
  [4261] = {x=608.677, y=-235.57, z=44, rx=-180, rz=165.18, shoulder=lefty, elbow=epositive, wrist=wpositive, fatherId=fReference[0]}
  [4262] = {x=610.067, y=-235.202, z=44, rx=-180, rz=165.007, shoulder=lefty, elbow=epositive, wrist=wpositive, fatherId=fReference[0]}
  [4263] = {x=611.457, y=-234.83, z=44, rx=-180, rz=164.835, shoulder=lefty, elbow=epositive, wrist=wpositive, fatherId=fReference[0]}
  [4264] = {x=612.846, y=-234.454, z=44, rx=-180, rz=164.664, shoulder=lefty, elbow=epositive, wrist=wpositive, fatherId=fReference[0]}
  [4265] = {x=614.235, y=-234.073, z=44, rx=-180, rz=164.493, shoulder=lefty, elbow=epositive, wrist=wpositive, fatherId=fReference[0]}
  [4266] = {x=615.623, y=-233.688, z=44, rx=180, rz=164.323, shoulder=lefty, elbow=epositive, wrist=wpositive, fatherId=fReference[0]}
  [4267] = {x=617.01, y=-233.298, z=44, rx=180, rz=164.153, shoulder=lefty, elbow=epositive, wrist=wpositive, fatherId=fReference[0]}
  [4268] = {x=618.397, y=-232.905, z=44, rx=180, rz=163.985, shoulder=lefty, elbow=epositive, wrist=wpositive, fatherId=fReference[0]}
  [4269] = {x=619.783, y=-232.507, z=44, rx=180, rz=163.816, shoulder=lefty, elbow=epositive, wrist=wpositive, fatherId=fReference[0]}
  [4270] = {x=621.169, y=-232.104, z=44, rx=180, rz=163.649, shoulder=lefty, elbow=epositive, wrist=wpositive, fatherId=fReference[0]}
  [4271] = {x=622.554, y=-231.698, z=44, rx=-180, rz=163.482, shoulder=lefty, elbow=epositive, wrist=wpositive, fatherId=fReference[0]}
  [4272] = {x=623.939, y=-231.288, z=44, rx=-180, rz=163.316, shoulder=lefty, elbow=epositive, wrist=wpositive, fatherId=fReference[0]}
  [4273] = {x=625.322, y=-230.873, z=44, rx=-180, rz=163.15, shoulder=lefty, elbow=epositive, wrist=wpositive, fatherId=fReference[0]}
  [4274] = {x=626.706, y=-230.454, z=44, rx=-180, rz=162.985, shoulder=lefty, elbow=epositive, wrist=wpositive, fatherId=fReference[0]}
  [4275] = {x=628.088, y=-230.031, z=44, rx=-180, rz=162.821, shoulder=lefty, elbow=epositive, wrist=wpositive, fatherId=fReference[0]}
  [4276] = {x=629.47, y=-229.604, z=44, rx=-180, rz=162.657, shoulder=lefty, elbow=epositive, wrist=wpositive, fatherId=fReference[0]}
  [4277] = {x=630.851, y=-229.172, z=44, rx=180, rz=162.494, shoulder=lefty, elbow=epositive, wrist=wpositive, fatherId=fReference[0]}
  [4278] = {x=632.232, y=-228.737, z=44, rx=180, rz=162.332, shoulder=lefty, elbow=epositive, wrist=wpositive, fatherId=fReference[0]}
  [4279] = {x=633.612, y=-228.297, z=44, rx=180, rz=162.171, shoulder=lefty, elbow=epositive, wrist=wpositive, fatherId=fReference[0]}
  [4280] = {x=634.991, y=-227.854, z=44, rx=-180, rz=162.01, shoulder=lefty, elbow=epositive, wrist=wpositive, fatherId=fReference[0]}
  [4281] = {x=636.37, y=-227.406, z=44, rx=180, rz=161.85, shoulder=lefty, elbow=epositive, wrist=wpositive, fatherId=fReference[0]}
  [4282] = {x=637.748, y=-226.954, z=44, rx=180, rz=161.69, shoulder=lefty, elbow=epositive, wrist=wpositive, fatherId=fReference[0]}
  [4283] = {x=639.125, y=-226.498, z=44, rx=-180, rz=161.531, shoulder=lefty, elbow=epositive, wrist=wpositive, fatherId=fReference[0]}
  [4284] = {x=640.502, y=-226.038, z=44, rx=-180, rz=161.373, shoulder=lefty, elbow=epositive, wrist=wpositive, fatherId=fReference[0]}
  [4285] = {x=641.878, y=-225.575, z=44, rx=-180, rz=161.216, shoulder=lefty, elbow=epositive, wrist=wpositive, fatherId=fReference[0]}
  [4286] = {x=643.254, y=-225.107, z=44, rx=-180, rz=161.059, shoulder=lefty, elbow=epositive, wrist=wpositive, fatherId=fReference[0]}
  [4287] = {x=644.628, y=-224.635, z=44, rx=-180, rz=160.903, shoulder=lefty, elbow=epositive, wrist=wpositive, fatherId=fReference[0]}
  [4288] = {x=646.002, y=-224.159, z=44, rx=-180, rz=160.748, shoulder=lefty, elbow=epositive, wrist=wpositive, fatherId=fReference[0]}
  [4289] = {x=647.376, y=-223.68, z=44, rx=180, rz=160.593, shoulder=lefty, elbow=epositive, wrist=wpositive, fatherId=fReference[0]}
  [4290] = {x=648.748, y=-223.196, z=44, rx=-180, rz=160.439, shoulder=lefty, elbow=epositive, wrist=wpositive, fatherId=fReference[0]}
  [4291] = {x=650.12, y=-222.709, z=44, rx=-180, rz=160.286, shoulder=lefty, elbow=epositive, wrist=wpositive, fatherId=fReference[0]}
  [4292] = {x=651.491, y=-222.217, z=44, rx=180, rz=160.133, shoulder=lefty, elbow=epositive, wrist=wpositive, fatherId=fReference[0]}
  [4293] = {x=652.862, y=-221.722, z=44, rx=-180, rz=159.981, shoulder=lefty, elbow=epositive, wrist=wpositive, fatherId=fReference[0]}
  [4294] = {x=654.232, y=-221.223, z=44, rx=-180, rz=159.83, shoulder=lefty, elbow=epositive, wrist=wpositive, fatherId=fReference[0]}
  [4295] = {x=655.601, y=-220.72, z=44, rx=-180, rz=159.68, shoulder=lefty, elbow=epositive, wrist=wpositive, fatherId=fReference[0]}
  [4296] = {x=656.969, y=-220.213, z=44, rx=-180, rz=159.53, shoulder=lefty, elbow=epositive, wrist=wpositive, fatherId=fReference[0]}
  [4297] = {x=658.337, y=-219.703, z=44, rx=-180, rz=159.381, shoulder=lefty, elbow=epositive, wrist=wpositive, fatherId=fReference[0]}
  [4298] = {x=659.704, y=-219.189, z=44, rx=180, rz=159.233, shoulder=lefty, elbow=epositive, wrist=wpositive, fatherId=fReference[0]}
  [4299] = {x=661.07, y=-218.67, z=44, rx=180, rz=159.086, shoulder=lefty, elbow=epositive, wrist=wpositive, fatherId=fReference[0]}
  [4300] = {x=662.436, y=-218.149, z=44, rx=180, rz=158.939, shoulder=lefty, elbow=epositive, wrist=wpositive, fatherId=fReference[0]}
  [4301] = {x=663.801, y=-217.623, z=44, rx=180, rz=158.793, shoulder=lefty, elbow=epositive, wrist=wpositive, fatherId=fReference[0]}
  [4302] = {x=665.165, y=-217.094, z=44, rx=-180, rz=158.647, shoulder=lefty, elbow=epositive, wrist=wpositive, fatherId=fReference[0]}
  [4303] = {x=666.528, y=-216.561, z=44, rx=180, rz=158.503, shoulder=lefty, elbow=epositive, wrist=wpositive, fatherId=fReference[0]}
  [4304] = {x=667.891, y=-216.024, z=44, rx=180, rz=158.359, shoulder=lefty, elbow=epositive, wrist=wpositive, fatherId=fReference[0]}
  [4305] = {x=669.253, y=-215.484, z=44, rx=-180, rz=158.216, shoulder=lefty, elbow=epositive, wrist=wpositive, fatherId=fReference[0]}
  [4306] = {x=670.614, y=-214.94, z=44, rx=-180, rz=158.073, shoulder=lefty, elbow=epositive, wrist=wpositive, fatherId=fReference[0]}
  [4307] = {x=671.974, y=-214.392, z=44, rx=180, rz=157.931, shoulder=lefty, elbow=epositive, wrist=wpositive, fatherId=fReference[0]}
  [4308] = {x=673.334, y=-213.841, z=44, rx=180, rz=157.79, shoulder=lefty, elbow=epositive, wrist=wpositive, fatherId=fReference[0]}
  [4309] = {x=674.693, y=-213.286, z=44, rx=-180, rz=157.65, shoulder=lefty, elbow=epositive, wrist=wpositive, fatherId=fReference[0]}
  [4310] = {x=676.052, y=-212.727, z=44, rx=-180, rz=157.51, shoulder=lefty, elbow=epositive, wrist=wpositive, fatherId=fReference[0]}
  [4311] = {x=677.409, y=-212.165, z=44, rx=-180, rz=157.371, shoulder=lefty, elbow=epositive, wrist=wpositive, fatherId=fReference[0]}
  [4312] = {x=678.766, y=-211.6, z=44, rx=180, rz=157.233, shoulder=lefty, elbow=epositive, wrist=wpositive, fatherId=fReference[0]}
  [4313] = {x=680.122, y=-211.031, z=44, rx=180, rz=157.096, shoulder=lefty, elbow=epositive, wrist=wpositive, fatherId=fReference[0]}
  [4314] = {x=681.477, y=-210.458, z=44, rx=180, rz=156.959, shoulder=lefty, elbow=epositive, wrist=wpositive, fatherId=fReference[0]}
  [4315] = {x=682.832, y=-209.882, z=44, rx=180, rz=156.823, shoulder=lefty, elbow=epositive, wrist=wpositive, fatherId=fReference[0]}
  [4316] = {x=684.186, y=-209.302, z=44, rx=-180, rz=156.688, shoulder=lefty, elbow=epositive, wrist=wpositive, fatherId=fReference[0]}
  [4317] = {x=685.539, y=-208.719, z=44, rx=180, rz=156.553, shoulder=lefty, elbow=epositive, wrist=wpositive, fatherId=fReference[0]}
  [4318] = {x=686.891, y=-208.133, z=44, rx=180, rz=156.42, shoulder=lefty, elbow=epositive, wrist=wpositive, fatherId=fReference[0]}
  [4319] = {x=688.243, y=-207.543, z=44, rx=-180, rz=156.287, shoulder=lefty, elbow=epositive, wrist=wpositive, fatherId=fReference[0]}
  [4320] = {x=689.593, y=-206.949, z=44, rx=180, rz=156.154, shoulder=lefty, elbow=epositive, wrist=wpositive, fatherId=fReference[0]}
  [4321] = {x=690.943, y=-206.353, z=44, rx=180, rz=156.023, shoulder=lefty, elbow=epositive, wrist=wpositive, fatherId=fReference[0]}
  [4322] = {x=692.293, y=-205.753, z=44, rx=180, rz=155.892, shoulder=lefty, elbow=epositive, wrist=wpositive, fatherId=fReference[0]}
  [4323] = {x=693.641, y=-205.149, z=44, rx=180, rz=155.762, shoulder=lefty, elbow=epositive, wrist=wpositive, fatherId=fReference[0]}
  [4324] = {x=694.989, y=-204.542, z=44, rx=180, rz=155.632, shoulder=lefty, elbow=epositive, wrist=wpositive, fatherId=fReference[0]}
  [4325] = {x=696.336, y=-203.932, z=44, rx=180, rz=155.503, shoulder=lefty, elbow=epositive, wrist=wpositive, fatherId=fReference[0]}
  [4326] = {x=697.682, y=-203.319, z=44, rx=180, rz=155.375, shoulder=lefty, elbow=epositive, wrist=wpositive, fatherId=fReference[0]}
  [4327] = {x=699.028, y=-202.702, z=44, rx=-180, rz=155.248, shoulder=lefty, elbow=epositive, wrist=wpositive, fatherId=fReference[0]}
  [4328] = {x=700.373, y=-202.082, z=44, rx=-180, rz=155.122, shoulder=lefty, elbow=epositive, wrist=wpositive, fatherId=fReference[0]}
  [4329] = {x=701.717, y=-201.459, z=44, rx=180, rz=154.996, shoulder=lefty, elbow=epositive, wrist=wpositive, fatherId=fReference[0]}
  [4330] = {x=703.06, y=-200.832, z=44, rx=180, rz=154.871, shoulder=lefty, elbow=epositive, wrist=wpositive, fatherId=fReference[0]}
  [4331] = {x=704.403, y=-200.203, z=44, rx=-180, rz=154.746, shoulder=lefty, elbow=epositive, wrist=wpositive, fatherId=fReference[0]}
  [4332] = {x=705.744, y=-199.57, z=44, rx=180, rz=154.622, shoulder=lefty, elbow=epositive, wrist=wpositive, fatherId=fReference[0]}
  [4333] = {x=707.085, y=-198.933, z=44, rx=-180, rz=154.499, shoulder=lefty, elbow=epositive, wrist=wpositive, fatherId=fReference[0]}
  [4334] = {x=708.426, y=-198.294, z=44, rx=180, rz=154.377, shoulder=lefty, elbow=epositive, wrist=wpositive, fatherId=fReference[0]}
  [4335] = {x=709.765, y=-197.652, z=44, rx=180, rz=154.256, shoulder=lefty, elbow=epositive, wrist=wpositive, fatherId=fReference[0]}
  [4336] = {x=711.104, y=-197.006, z=44, rx=180, rz=154.135, shoulder=lefty, elbow=epositive, wrist=wpositive, fatherId=fReference[0]}
  [4337] = {x=712.442, y=-196.357, z=44, rx=180, rz=154.015, shoulder=lefty, elbow=epositive, wrist=wpositive, fatherId=fReference[0]}
  [4338] = {x=713.779, y=-195.706, z=44, rx=180, rz=153.895, shoulder=lefty, elbow=epositive, wrist=wpositive, fatherId=fReference[0]}
  [4339] = {x=715.116, y=-195.051, z=44, rx=-180, rz=153.776, shoulder=lefty, elbow=epositive, wrist=wpositive, fatherId=fReference[0]}
  [4340] = {x=716.452, y=-194.393, z=44, rx=180, rz=153.658, shoulder=lefty, elbow=epositive, wrist=wpositive, fatherId=fReference[0]}
  [4341] = {x=717.787, y=-193.732, z=44, rx=-180, rz=153.541, shoulder=lefty, elbow=epositive, wrist=wpositive, fatherId=fReference[0]}
  [4342] = {x=719.121, y=-193.067, z=44, rx=-180, rz=153.424, shoulder=lefty, elbow=epositive, wrist=wpositive, fatherId=fReference[0]}
  [4343] = {x=720.455, y=-192.4, z=44, rx=180, rz=153.309, shoulder=lefty, elbow=epositive, wrist=wpositive, fatherId=fReference[0]}
  [4344] = {x=721.788, y=-191.73, z=44, rx=180, rz=153.193, shoulder=lefty, elbow=epositive, wrist=wpositive, fatherId=fReference[0]}
  [4345] = {x=723.12, y=-191.057, z=44, rx=180, rz=153.079, shoulder=lefty, elbow=epositive, wrist=wpositive, fatherId=fReference[0]}
  [4346] = {x=724.451, y=-190.381, z=44, rx=180, rz=152.965, shoulder=lefty, elbow=epositive, wrist=wpositive, fatherId=fReference[0]}
  [4347] = {x=725.782, y=-189.702, z=44, rx=180, rz=152.852, shoulder=lefty, elbow=epositive, wrist=wpositive, fatherId=fReference[0]}
  [4348] = {x=727.112, y=-189.02, z=44, rx=180, rz=152.739, shoulder=lefty, elbow=epositive, wrist=wpositive, fatherId=fReference[0]}
  [4349] = {x=728.441, y=-188.335, z=44, rx=-180, rz=152.628, shoulder=lefty, elbow=epositive, wrist=wpositive, fatherId=fReference[0]}
  [4350] = {x=729.77, y=-187.647, z=44, rx=180, rz=152.517, shoulder=lefty, elbow=epositive, wrist=wpositive, fatherId=fReference[0]}
  [4351] = {x=731.098, y=-186.957, z=44, rx=180, rz=152.406, shoulder=lefty, elbow=epositive, wrist=wpositive, fatherId=fReference[0]}
  [4352] = {x=732.425, y=-186.263, z=44, rx=-180, rz=152.297, shoulder=lefty, elbow=epositive, wrist=wpositive, fatherId=fReference[0]}
  [4353] = {x=733.751, y=-185.567, z=44, rx=-180, rz=152.188, shoulder=lefty, elbow=epositive, wrist=wpositive, fatherId=fReference[0]}
  [4354] = {x=735.077, y=-184.867, z=44, rx=-180, rz=152.079, shoulder=lefty, elbow=epositive, wrist=wpositive, fatherId=fReference[0]}
  [4355] = {x=736.401, y=-184.165, z=44, rx=-180, rz=151.972, shoulder=lefty, elbow=epositive, wrist=wpositive, fatherId=fReference[0]}
  [4356] = {x=737.726, y=-183.46, z=44, rx=180, rz=151.865, shoulder=lefty, elbow=epositive, wrist=wpositive, fatherId=fReference[0]}
  [4357] = {x=739.049, y=-182.753, z=44, rx=180, rz=151.759, shoulder=lefty, elbow=epositive, wrist=wpositive, fatherId=fReference[0]}
  [4358] = {x=740.372, y=-182.042, z=44, rx=-180, rz=151.653, shoulder=lefty, elbow=epositive, wrist=wpositive, fatherId=fReference[0]}
  [4359] = {x=741.694, y=-181.329, z=44, rx=-180, rz=151.548, shoulder=lefty, elbow=epositive, wrist=wpositive, fatherId=fReference[0]}
  [4360] = {x=743.015, y=-180.613, z=44, rx=-180, rz=151.444, shoulder=lefty, elbow=epositive, wrist=wpositive, fatherId=fReference[0]}
  [4361] = {x=744.336, y=-179.894, z=44, rx=180, rz=151.341, shoulder=lefty, elbow=epositive, wrist=wpositive, fatherId=fReference[0]}
  [4362] = {x=745.656, y=-179.173, z=44, rx=-180, rz=151.238, shoulder=lefty, elbow=epositive, wrist=wpositive, fatherId=fReference[0]}
  [4363] = {x=746.975, y=-178.449, z=44, rx=-180, rz=151.136, shoulder=lefty, elbow=epositive, wrist=wpositive, fatherId=fReference[0]}
  [4364] = {x=748.293, y=-177.722, z=44, rx=180, rz=151.034, shoulder=lefty, elbow=epositive, wrist=wpositive, fatherId=fReference[0]}
  [4365] = {x=749.611, y=-176.993, z=44, rx=180, rz=150.933, shoulder=lefty, elbow=epositive, wrist=wpositive, fatherId=fReference[0]}
  [4366] = {x=750.928, y=-176.26, z=44, rx=-180, rz=150.833, shoulder=lefty, elbow=epositive, wrist=wpositive, fatherId=fReference[0]}
  [4367] = {x=752.244, y=-175.526, z=44, rx=-180, rz=150.734, shoulder=lefty, elbow=epositive, wrist=wpositive, fatherId=fReference[0]}
  [4368] = {x=753.56, y=-174.788, z=44, rx=180, rz=150.635, shoulder=lefty, elbow=epositive, wrist=wpositive, fatherId=fReference[0]}
  [4369] = {x=754.875, y=-174.049, z=44, rx=-180, rz=150.537, shoulder=lefty, elbow=epositive, wrist=wpositive, fatherId=fReference[0]}
  [4370] = {x=756.189, y=-173.306, z=44, rx=180, rz=150.439, shoulder=lefty, elbow=epositive, wrist=wpositive, fatherId=fReference[0]}
  [4371] = {x=757.503, y=-172.561, z=44, rx=180, rz=150.342, shoulder=lefty, elbow=epositive, wrist=wpositive, fatherId=fReference[0]}
  [4372] = {x=758.816, y=-171.814, z=44, rx=-180, rz=150.246, shoulder=lefty, elbow=epositive, wrist=wpositive, fatherId=fReference[0]}
  [4373] = {x=760.128, y=-171.064, z=44, rx=-180, rz=150.151, shoulder=lefty, elbow=epositive, wrist=wpositive, fatherId=fReference[0]}
  [4374] = {x=761.439, y=-170.311, z=44, rx=180, rz=150.056, shoulder=lefty, elbow=epositive, wrist=wpositive, fatherId=fReference[0]}
  [4375] = {x=762.75, y=-169.556, z=44, rx=180, rz=149.961, shoulder=lefty, elbow=epositive, wrist=wpositive, fatherId=fReference[0]}
  [4376] = {x=764.06, y=-168.798, z=44, rx=180, rz=149.868, shoulder=lefty, elbow=epositive, wrist=wpositive, fatherId=fReference[0]}
  [4377] = {x=765.369, y=-168.038, z=44, rx=-180, rz=149.775, shoulder=lefty, elbow=epositive, wrist=wpositive, fatherId=fReference[0]}
  [4378] = {x=766.678, y=-167.276, z=44, rx=180, rz=149.683, shoulder=lefty, elbow=epositive, wrist=wpositive, fatherId=fReference[0]}
  [4379] = {x=767.986, y=-166.511, z=44, rx=-180, rz=149.591, shoulder=lefty, elbow=epositive, wrist=wpositive, fatherId=fReference[0]}
  [4380] = {x=769.293, y=-165.744, z=44, rx=180, rz=149.5, shoulder=lefty, elbow=epositive, wrist=wpositive, fatherId=fReference[0]}
  [4381] = {x=770.6, y=-164.974, z=44, rx=-180, rz=149.41, shoulder=lefty, elbow=epositive, wrist=wpositive, fatherId=fReference[0]}
  [4382] = {x=771.906, y=-164.202, z=44, rx=180, rz=149.32, shoulder=lefty, elbow=epositive, wrist=wpositive, fatherId=fReference[0]}
  [4383] = {x=773.211, y=-163.428, z=44, rx=180, rz=149.231, shoulder=lefty, elbow=epositive, wrist=wpositive, fatherId=fReference[0]}
  [4384] = {x=774.516, y=-162.651, z=44, rx=-180, rz=149.142, shoulder=lefty, elbow=epositive, wrist=wpositive, fatherId=fReference[0]}
  [4385] = {x=775.82, y=-161.872, z=44, rx=180, rz=149.054, shoulder=lefty, elbow=epositive, wrist=wpositive, fatherId=fReference[0]}
  [4386] = {x=777.123, y=-161.091, z=44, rx=-180, rz=148.967, shoulder=lefty, elbow=epositive, wrist=wpositive, fatherId=fReference[0]}
  [4387] = {x=778.425, y=-160.307, z=44, rx=-180, rz=148.881, shoulder=lefty, elbow=epositive, wrist=wpositive, fatherId=fReference[0]}
  [4388] = {x=779.727, y=-159.521, z=44, rx=180, rz=148.795, shoulder=lefty, elbow=epositive, wrist=wpositive, fatherId=fReference[0]}
  [4389] = {x=781.028, y=-158.733, z=44, rx=-180, rz=148.709, shoulder=lefty, elbow=epositive, wrist=wpositive, fatherId=fReference[0]}
  [4390] = {x=782.329, y=-157.942, z=44, rx=-180, rz=148.625, shoulder=lefty, elbow=epositive, wrist=wpositive, fatherId=fReference[0]}
  [4391] = {x=783.629, y=-157.15, z=44, rx=180, rz=148.54, shoulder=lefty, elbow=epositive, wrist=wpositive, fatherId=fReference[0]}
  [4392] = {x=784.928, y=-156.355, z=44, rx=180, rz=148.457, shoulder=lefty, elbow=epositive, wrist=wpositive, fatherId=fReference[0]}
  [4393] = {x=786.227, y=-155.558, z=44, rx=180, rz=148.374, shoulder=lefty, elbow=epositive, wrist=wpositive, fatherId=fReference[0]}
  [4394] = {x=787.524, y=-154.758, z=44, rx=180, rz=148.292, shoulder=lefty, elbow=epositive, wrist=wpositive, fatherId=fReference[0]}
  [4395] = {x=788.822, y=-153.957, z=44, rx=-180, rz=148.21, shoulder=lefty, elbow=epositive, wrist=wpositive, fatherId=fReference[0]}
  [4396] = {x=790.118, y=-153.153, z=44, rx=180, rz=148.129, shoulder=lefty, elbow=epositive, wrist=wpositive, fatherId=fReference[0]}
  [4397] = {x=791.414, y=-152.348, z=44, rx=-180, rz=148.049, shoulder=lefty, elbow=epositive, wrist=wpositive, fatherId=fReference[0]}
  [4398] = {x=792.709, y=-151.54, z=44, rx=-180, rz=147.969, shoulder=lefty, elbow=epositive, wrist=wpositive, fatherId=fReference[0]}
  [4399] = {x=794.004, y=-150.73, z=44, rx=-180, rz=147.89, shoulder=lefty, elbow=epositive, wrist=wpositive, fatherId=fReference[0]}
  [4400] = {x=795.298, y=-149.918, z=44, rx=-180, rz=147.811, shoulder=lefty, elbow=epositive, wrist=wpositive, fatherId=fReference[0]}
  [4401] = {x=796.591, y=-149.104, z=44, rx=-180, rz=147.733, shoulder=lefty, elbow=epositive, wrist=wpositive, fatherId=fReference[0]}
  [4402] = {x=797.884, y=-148.288, z=44, rx=-180, rz=147.656, shoulder=lefty, elbow=epositive, wrist=wpositive, fatherId=fReference[0]}
  [4403] = {x=799.175, y=-147.47, z=44, rx=-180, rz=147.579, shoulder=lefty, elbow=epositive, wrist=wpositive, fatherId=fReference[0]}
  [4404] = {x=800.467, y=-146.65, z=44, rx=180, rz=147.503, shoulder=lefty, elbow=epositive, wrist=wpositive, fatherId=fReference[0]}
  [4405] = {x=801.757, y=-145.827, z=44, rx=-180, rz=147.427, shoulder=lefty, elbow=epositive, wrist=wpositive, fatherId=fReference[0]}
  [4406] = {x=803.047, y=-145.003, z=44, rx=180, rz=147.352, shoulder=lefty, elbow=epositive, wrist=wpositive, fatherId=fReference[0]}
  [4407] = {x=804.337, y=-144.177, z=44, rx=180, rz=147.277, shoulder=lefty, elbow=epositive, wrist=wpositive, fatherId=fReference[0]}
  [4408] = {x=805.626, y=-143.349, z=44, rx=-180, rz=147.204, shoulder=lefty, elbow=epositive, wrist=wpositive, fatherId=fReference[0]}
  [4409] = {x=806.914, y=-142.519, z=44, rx=180, rz=147.13, shoulder=lefty, elbow=epositive, wrist=wpositive, fatherId=fReference[0]}
  [4410] = {x=808.201, y=-141.687, z=44, rx=-180, rz=147.058, shoulder=lefty, elbow=epositive, wrist=wpositive, fatherId=fReference[0]}
  [4411] = {x=809.488, y=-140.853, z=44, rx=-180, rz=146.986, shoulder=lefty, elbow=epositive, wrist=wpositive, fatherId=fReference[0]}
  [4412] = {x=810.774, y=-140.017, z=44, rx=-180, rz=146.914, shoulder=lefty, elbow=epositive, wrist=wpositive, fatherId=fReference[0]}
  [4413] = {x=812.06, y=-139.18, z=44, rx=-180, rz=146.843, shoulder=lefty, elbow=epositive, wrist=wpositive, fatherId=fReference[0]}
  [4414] = {x=813.345, y=-138.34, z=44, rx=180, rz=146.773, shoulder=lefty, elbow=epositive, wrist=wpositive, fatherId=fReference[0]}
  [4415] = {x=814.629, y=-137.499, z=44, rx=-180, rz=146.703, shoulder=lefty, elbow=epositive, wrist=wpositive, fatherId=fReference[0]}
  [4416] = {x=815.913, y=-136.656, z=44, rx=180, rz=146.634, shoulder=lefty, elbow=epositive, wrist=wpositive, fatherId=fReference[0]}
  [4417] = {x=817.196, y=-135.811, z=44, rx=180, rz=146.565, shoulder=lefty, elbow=epositive, wrist=wpositive, fatherId=fReference[0]}
  [4418] = {x=818.479, y=-134.964, z=44, rx=-180, rz=146.497, shoulder=lefty, elbow=epositive, wrist=wpositive, fatherId=fReference[0]}
  [4419] = {x=819.761, y=-134.115, z=44, rx=180, rz=146.429, shoulder=lefty, elbow=epositive, wrist=wpositive, fatherId=fReference[0]}
  [4420] = {x=821.042, y=-133.265, z=44, rx=-180, rz=146.362, shoulder=lefty, elbow=epositive, wrist=wpositive, fatherId=fReference[0]}
  [4421] = {x=822.323, y=-132.413, z=44, rx=180, rz=146.296, shoulder=lefty, elbow=epositive, wrist=wpositive, fatherId=fReference[0]}
  [4422] = {x=823.603, y=-131.559, z=44, rx=180, rz=146.23, shoulder=lefty, elbow=epositive, wrist=wpositive, fatherId=fReference[0]}
  [4423] = {x=824.882, y=-130.703, z=44, rx=180, rz=146.165, shoulder=lefty, elbow=epositive, wrist=wpositive, fatherId=fReference[0]}
  [4424] = {x=826.161, y=-129.846, z=44, rx=-180, rz=146.1, shoulder=lefty, elbow=epositive, wrist=wpositive, fatherId=fReference[0]}
  [4425] = {x=827.44, y=-128.987, z=44, rx=180, rz=146.036, shoulder=lefty, elbow=epositive, wrist=wpositive, fatherId=fReference[0]}
  [4426] = {x=828.717, y=-128.127, z=44, rx=-180, rz=145.972, shoulder=lefty, elbow=epositive, wrist=wpositive, fatherId=fReference[0]}
  [4427] = {x=829.994, y=-127.264, z=44, rx=180, rz=145.909, shoulder=lefty, elbow=epositive, wrist=wpositive, fatherId=fReference[0]}
  [4428] = {x=831.271, y=-126.4, z=44, rx=180, rz=145.847, shoulder=lefty, elbow=epositive, wrist=wpositive, fatherId=fReference[0]}
  [4429] = {x=832.547, y=-125.535, z=44, rx=180, rz=145.785, shoulder=lefty, elbow=epositive, wrist=wpositive, fatherId=fReference[0]}
  [4430] = {x=833.822, y=-124.667, z=44, rx=-180, rz=145.723, shoulder=lefty, elbow=epositive, wrist=wpositive, fatherId=fReference[0]}
  [4431] = {x=835.097, y=-123.798, z=44, rx=-180, rz=145.662, shoulder=lefty, elbow=epositive, wrist=wpositive, fatherId=fReference[0]}
  [4432] = {x=836.372, y=-122.928, z=44, rx=180, rz=145.602, shoulder=lefty, elbow=epositive, wrist=wpositive, fatherId=fReference[0]}
  [4433] = {x=837.645, y=-122.056, z=44, rx=-180, rz=145.542, shoulder=lefty, elbow=epositive, wrist=wpositive, fatherId=fReference[0]}
  [4434] = {x=838.918, y=-121.182, z=44, rx=-180, rz=145.483, shoulder=lefty, elbow=epositive, wrist=wpositive, fatherId=fReference[0]}
  [4435] = {x=840.191, y=-120.307, z=44, rx=180, rz=145.424, shoulder=lefty, elbow=epositive, wrist=wpositive, fatherId=fReference[0]}
  [4436] = {x=841.463, y=-119.43, z=44, rx=180, rz=145.366, shoulder=lefty, elbow=epositive, wrist=wpositive, fatherId=fReference[0]}
  [4437] = {x=842.734, y=-118.552, z=44, rx=180, rz=145.308, shoulder=lefty, elbow=epositive, wrist=wpositive, fatherId=fReference[0]}
  [4438] = {x=844.005, y=-117.672, z=44, rx=180, rz=145.251, shoulder=lefty, elbow=epositive, wrist=wpositive, fatherId=fReference[0]}
  [4439] = {x=845.276, y=-116.791, z=44, rx=180, rz=145.195, shoulder=lefty, elbow=epositive, wrist=wpositive, fatherId=fReference[0]}
  [4440] = {x=846.545, y=-115.908, z=44, rx=180, rz=145.139, shoulder=lefty, elbow=epositive, wrist=wpositive, fatherId=fReference[0]}
  [4441] = {x=847.815, y=-115.024, z=44, rx=180, rz=145.083, shoulder=lefty, elbow=epositive, wrist=wpositive, fatherId=fReference[0]}
  [4442] = {x=849.084, y=-114.139, z=44, rx=180, rz=145.028, shoulder=lefty, elbow=epositive, wrist=wpositive, fatherId=fReference[0]}
  [4443] = {x=850.352, y=-113.251, z=44, rx=180, rz=144.974, shoulder=lefty, elbow=epositive, wrist=wpositive, fatherId=fReference[0]}
  [4444] = {x=851.619, y=-112.363, z=44, rx=180, rz=144.92, shoulder=lefty, elbow=epositive, wrist=wpositive, fatherId=fReference[0]}
  [4445] = {x=852.887, y=-111.473, z=44, rx=-180, rz=144.866, shoulder=lefty, elbow=epositive, wrist=wpositive, fatherId=fReference[0]}
  [4446] = {x=854.153, y=-110.582, z=44, rx=180, rz=144.813, shoulder=lefty, elbow=epositive, wrist=wpositive, fatherId=fReference[0]}
  [4447] = {x=855.419, y=-109.689, z=44, rx=180, rz=144.761, shoulder=lefty, elbow=epositive, wrist=wpositive, fatherId=fReference[0]}
  [4448] = {x=856.685, y=-108.795, z=44, rx=-180, rz=144.709, shoulder=lefty, elbow=epositive, wrist=wpositive, fatherId=fReference[0]}
  [4449] = {x=857.95, y=-107.899, z=44, rx=180, rz=144.657, shoulder=lefty, elbow=epositive, wrist=wpositive, fatherId=fReference[0]}
  [4450] = {x=859.215, y=-107.003, z=44, rx=-180, rz=144.607, shoulder=lefty, elbow=epositive, wrist=wpositive, fatherId=fReference[0]}
  [4451] = {x=860.479, y=-106.104, z=44, rx=-180, rz=144.556, shoulder=lefty, elbow=epositive, wrist=wpositive, fatherId=fReference[0]}
  [4452] = {x=861.742, y=-105.205, z=44, rx=-180, rz=144.506, shoulder=lefty, elbow=epositive, wrist=wpositive, fatherId=fReference[0]}
  [4453] = {x=863.006, y=-104.304, z=44, rx=180, rz=144.457, shoulder=lefty, elbow=epositive, wrist=wpositive, fatherId=fReference[0]}
  [4454] = {x=864.268, y=-103.402, z=44, rx=180, rz=144.408, shoulder=lefty, elbow=epositive, wrist=wpositive, fatherId=fReference[0]}
  [4455] = {x=865.53, y=-102.499, z=44, rx=180, rz=144.36, shoulder=lefty, elbow=epositive, wrist=wpositive, fatherId=fReference[0]}
  [4456] = {x=866.792, y=-101.594, z=44, rx=180, rz=144.312, shoulder=lefty, elbow=epositive, wrist=wpositive, fatherId=fReference[0]}
  [4457] = {x=868.053, y=-100.688, z=44, rx=-180, rz=144.265, shoulder=lefty, elbow=epositive, wrist=wpositive, fatherId=fReference[0]}
  [4458] = {x=869.314, y=-99.781, z=44, rx=180, rz=144.218, shoulder=lefty, elbow=epositive, wrist=wpositive, fatherId=fReference[0]}
  [4459] = {x=870.574, y=-98.873, z=44, rx=-180, rz=144.172, shoulder=lefty, elbow=epositive, wrist=wpositive, fatherId=fReference[0]}
  [4460] = {x=871.834, y=-97.963, z=44, rx=-180, rz=144.126, shoulder=lefty, elbow=epositive, wrist=wpositive, fatherId=fReference[0]}
  [4461] = {x=873.094, y=-97.052, z=44, rx=180, rz=144.08, shoulder=lefty, elbow=epositive, wrist=wpositive, fatherId=fReference[0]}
  [4462] = {x=874.353, y=-96.14, z=44, rx=180, rz=144.036, shoulder=lefty, elbow=epositive, wrist=wpositive, fatherId=fReference[0]}
  [4463] = {x=875.611, y=-95.227, z=44, rx=180, rz=143.991, shoulder=lefty, elbow=epositive, wrist=wpositive, fatherId=fReference[0]}
  [4464] = {x=876.869, y=-94.313, z=44, rx=180, rz=143.947, shoulder=lefty, elbow=epositive, wrist=wpositive, fatherId=fReference[0]}
  [4465] = {x=878.127, y=-93.397, z=44, rx=-180, rz=143.904, shoulder=lefty, elbow=epositive, wrist=wpositive, fatherId=fReference[0]}
  [4466] = {x=879.384, y=-92.481, z=44, rx=-180, rz=143.861, shoulder=lefty, elbow=epositive, wrist=wpositive, fatherId=fReference[0]}
  [4467] = {x=880.641, y=-91.563, z=44, rx=180, rz=143.819, shoulder=lefty, elbow=epositive, wrist=wpositive, fatherId=fReference[0]}
  [4468] = {x=881.897, y=-90.644, z=44, rx=180, rz=143.777, shoulder=lefty, elbow=epositive, wrist=wpositive, fatherId=fReference[0]}
  [4469] = {x=883.153, y=-89.724, z=44, rx=-180, rz=143.735, shoulder=lefty, elbow=epositive, wrist=wpositive, fatherId=fReference[0]}
  [4470] = {x=884.409, y=-88.803, z=44, rx=180, rz=143.694, shoulder=lefty, elbow=epositive, wrist=wpositive, fatherId=fReference[0]}
  [4471] = {x=885.664, y=-87.881, z=44, rx=180, rz=143.654, shoulder=lefty, elbow=epositive, wrist=wpositive, fatherId=fReference[0]}
  [4472] = {x=886.919, y=-86.957, z=44, rx=180, rz=143.614, shoulder=lefty, elbow=epositive, wrist=wpositive, fatherId=fReference[0]}
  [4473] = {x=888.173, y=-86.033, z=44, rx=-180, rz=143.574, shoulder=lefty, elbow=epositive, wrist=wpositive, fatherId=fReference[0]}
  [4474] = {x=889.427, y=-85.108, z=44, rx=180, rz=143.535, shoulder=lefty, elbow=epositive, wrist=wpositive, fatherId=fReference[0]}
  [4475] = {x=890.681, y=-84.181, z=44, rx=-180, rz=143.497, shoulder=lefty, elbow=epositive, wrist=wpositive, fatherId=fReference[0]}
  [4476] = {x=891.934, y=-83.254, z=44, rx=180, rz=143.459, shoulder=lefty, elbow=epositive, wrist=wpositive, fatherId=fReference[0]}
  [4477] = {x=893.187, y=-82.325, z=44, rx=180, rz=143.421, shoulder=lefty, elbow=epositive, wrist=wpositive, fatherId=fReference[0]}
  [4478] = {x=894.439, y=-81.396, z=44, rx=180, rz=143.384, shoulder=lefty, elbow=epositive, wrist=wpositive, fatherId=fReference[0]}
  [4479] = {x=895.691, y=-80.465, z=44, rx=180, rz=143.347, shoulder=lefty, elbow=epositive, wrist=wpositive, fatherId=fReference[0]}
  [4480] = {x=896.943, y=-79.534, z=44, rx=180, rz=143.311, shoulder=lefty, elbow=epositive, wrist=wpositive, fatherId=fReference[0]}
  [4481] = {x=898.195, y=-78.602, z=44, rx=180, rz=143.275, shoulder=lefty, elbow=epositive, wrist=wpositive, fatherId=fReference[0]}
  [4482] = {x=899.446, y=-77.668, z=44, rx=180, rz=143.24, shoulder=lefty, elbow=epositive, wrist=wpositive, fatherId=fReference[0]}
  [4483] = {x=900.696, y=-76.734, z=44, rx=180, rz=143.205, shoulder=lefty, elbow=epositive, wrist=wpositive, fatherId=fReference[0]}
  [4484] = {x=901.947, y=-75.799, z=44, rx=-180, rz=143.171, shoulder=lefty, elbow=epositive, wrist=wpositive, fatherId=fReference[0]}
  [4485] = {x=903.197, y=-74.862, z=44, rx=-180, rz=143.137, shoulder=lefty, elbow=epositive, wrist=wpositive, fatherId=fReference[0]}
  [4486] = {x=904.447, y=-73.925, z=44, rx=-180, rz=143.103, shoulder=lefty, elbow=epositive, wrist=wpositive, fatherId=fReference[0]}
  [4487] = {x=905.696, y=-72.987, z=44, rx=-180, rz=143.07, shoulder=lefty, elbow=epositive, wrist=wpositive, fatherId=fReference[0]}
  [4488] = {x=906.945, y=-72.049, z=44, rx=180, rz=143.038, shoulder=lefty, elbow=epositive, wrist=wpositive, fatherId=fReference[0]}
  [4489] = {x=908.194, y=-71.109, z=44, rx=-180, rz=143.006, shoulder=lefty, elbow=epositive, wrist=wpositive, fatherId=fReference[0]}
  [4490] = {x=909.442, y=-70.168, z=44, rx=-180, rz=142.974, shoulder=lefty, elbow=epositive, wrist=wpositive, fatherId=fReference[0]}
  [4491] = {x=910.69, y=-69.227, z=44, rx=-180, rz=142.943, shoulder=lefty, elbow=epositive, wrist=wpositive, fatherId=fReference[0]}
  [4492] = {x=911.938, y=-68.285, z=44, rx=180, rz=142.912, shoulder=lefty, elbow=epositive, wrist=wpositive, fatherId=fReference[0]}
  [4493] = {x=913.185, y=-67.342, z=44, rx=180, rz=142.882, shoulder=lefty, elbow=epositive, wrist=wpositive, fatherId=fReference[0]}
  [4494] = {x=914.433, y=-66.398, z=44, rx=180, rz=142.853, shoulder=lefty, elbow=epositive, wrist=wpositive, fatherId=fReference[0]}
  [4495] = {x=915.68, y=-65.453, z=44, rx=180, rz=142.823, shoulder=lefty, elbow=epositive, wrist=wpositive, fatherId=fReference[0]}
  [4496] = {x=916.926, y=-64.508, z=44, rx=-180, rz=142.794, shoulder=lefty, elbow=epositive, wrist=wpositive, fatherId=fReference[0]}
  [4497] = {x=918.172, y=-63.562, z=44, rx=180, rz=142.766, shoulder=lefty, elbow=epositive, wrist=wpositive, fatherId=fReference[0]}
  [4498] = {x=919.418, y=-62.615, z=44, rx=-180, rz=142.738, shoulder=lefty, elbow=epositive, wrist=wpositive, fatherId=fReference[0]}
  [4499] = {x=920.664, y=-61.667, z=44, rx=-180, rz=142.71, shoulder=lefty, elbow=epositive, wrist=wpositive, fatherId=fReference[0]}
  [4500] = {x=921.91, y=-60.719, z=44, rx=-180, rz=142.683, shoulder=lefty, elbow=epositive, wrist=wpositive, fatherId=fReference[0]}
  [4501] = {x=923.155, y=-59.769, z=44, rx=-180, rz=142.657, shoulder=lefty, elbow=epositive, wrist=wpositive, fatherId=fReference[0]}
  [4502] = {x=924.4, y=-58.82, z=44, rx=180, rz=142.631, shoulder=lefty, elbow=epositive, wrist=wpositive, fatherId=fReference[0]}
  [4503] = {x=925.644, y=-57.869, z=44, rx=-180, rz=142.605, shoulder=lefty, elbow=epositive, wrist=wpositive, fatherId=fReference[0]}
  [4504] = {x=926.889, y=-56.918, z=44, rx=180, rz=142.58, shoulder=lefty, elbow=epositive, wrist=wpositive, fatherId=fReference[0]}
  [4505] = {x=928.133, y=-55.966, z=44, rx=-180, rz=142.555, shoulder=lefty, elbow=epositive, wrist=wpositive, fatherId=fReference[0]}
  [4506] = {x=929.377, y=-55.013, z=44, rx=180, rz=142.53, shoulder=lefty, elbow=epositive, wrist=wpositive, fatherId=fReference[0]}
  [4507] = {x=930.621, y=-54.06, z=44, rx=-180, rz=142.507, shoulder=lefty, elbow=epositive, wrist=wpositive, fatherId=fReference[0]}
  [4508] = {x=931.864, y=-53.106, z=44, rx=-180, rz=142.483, shoulder=lefty, elbow=epositive, wrist=wpositive, fatherId=fReference[0]}
